// TIA Portal V20 export
FUNCTION_BLOCK "Sequence_3_TopTapeFixStage"   // FB32850, LAD
TITLE = Sequence
// Sequence template programmend in ladder logic
// stored: IsIECCheckEnabled true, MemoryReserve 100, Namespace Unit1.Em3, SetENOAutomatically true
   VAR_INPUT
      unitStatus : "LAF_typeUnitStatus";
   END_VAR
   VAR
      instSequenceLADControl { ExternalWritable := 'False'} : "LAF_ControlLadSequence";
      instSequenceLADStatus { ExternalWritable := 'False'} : "LAF_StatusLadSequence";
      statTonTime { ExternalWritable := 'False'} : Array[0..9999] of TON_TIME;
   END_VAR
   VAR_TEMP
      tempCustomerAction : Bool;   // Placeholder for possible actions
      tempDo_nothing_and_wait_for_init : Bool;   // Placeholder for doing nothing
      tempSafeStateCondition : Bool;   // Temp Condition for the equipment module to be in a safe state
   END_VAR
   VAR CONSTANT
      delayTime : Time := T#100ms;
      STEP_IDLE : DInt := 1;
      JOB_1_STEP_01 : DInt := 101;
      JOB_1_STEP_10 : DInt := 110;
      JOB_1_STEP_11 : DInt := 111;
      JOB_1_STEP_20 : DInt := 120;
      JOB_1_STEP_21 : DInt := 121;
      JOB_1_STEP_30 : DInt := 130;
      JOB_1_STEP_40 : DInt := 140;
      JOB_1_STEP_50 : DInt := 150;
      JOB_1_STEP_60 : DInt := 160;
      JOB_1_STEP_70 : DInt := 170;
      JOB_1_STEP_80 : DInt := 180;
      JOB_1_STEP_90 : DInt := 190;
      JOB_2_STEP_01 : DInt := 201;
      JOB_2_STEP_10 : DInt := 210;
      JOB_2_STEP_20 : DInt := 220;
      JOB_2_STEP_30 : DInt := 230;
      JOB_2_STEP_31 : DInt := 231;
      JOB_2_STEP_32 : DInt := 232;
      JOB_2_STEP_33 : DInt := 233;
      JOB_2_STEP_40 : DInt := 240;
      JOB_2_STEP_50 : DInt := 250;
      JOB_2_STEP_51 : DInt := 250;
      JOB_2_STEP_60 : DInt := 260;
      JOB_2_STEP_70 : DInt := 270;
      JOB_2_STEP_80 : DInt := 280;
      JOB_2_STEP_81 : DInt := 281;
      JOB_2_STEP_90 : DInt := 290;
      JOB_3_STEP_01 : DInt := 301;
      JOB_3_STEP_10 : DInt := 310;
      JOB_3_STEP_20 : DInt := 320;
      JOB_3_STEP_30 : DInt := 330;
      JOB_3_STEP_40 : DInt := 340;
      JOB_3_STEP_50 : DInt := 350;
      JOB_3_STEP_60 : DInt := 360;
      JOB_3_STEP_61 : DInt := 361;
      JOB_3_STEP_70 : DInt := 370;
      JOB_3_STEP_80 : DInt := 380;
      JOB_3_STEP_90 : DInt := 390;
      JOB_4_STEP_01 : DInt := 401;
      JOB_4_STEP_10 : DInt := 410;
      JOB_4_STEP_20 : DInt := 420;
      JOB_4_STEP_30 : DInt := 430;
      JOB_4_STEP_31 : DInt := 431;
      JOB_4_STEP_32 : DInt := 432;
      JOB_4_STEP_40 : DInt := 440;
      JOB_4_STEP_41 : DInt := 441;
      JOB_4_STEP_50 : DInt := 450;
      JOB_4_STEP_60 : DInt := 460;
      JOB_4_STEP_70 : DInt := 470;
      JOB_4_STEP_80 : DInt := 480;
      JOB_4_STEP_90 : DInt := 490;
      JOB_5_STEP_01 : DInt := 501;
      JOB_5_STEP_10 : DInt := 510;
      JOB_5_STEP_20 : DInt := 520;
      JOB_5_STEP_30 : DInt := 530;
      JOB_5_STEP_31 : DInt := 531;
      JOB_5_STEP_32 : DInt := 532;
      JOB_5_STEP_40 : DInt := 540;
      JOB_5_STEP_50 : DInt := 550;
      JOB_5_STEP_60 : DInt := 560;
      JOB_5_STEP_70 : DInt := 570;
      JOB_5_STEP_80 : DInt := 580;
      JOB_5_STEP_90 : DInt := 590;
      STEP_IMMEDIATE_STOP : DInt := 9001;   // Step executed when an immediate stop command is triggered for the sequence (i.e. when unit is in state aborting)
      TO_DO_INSERT_ACTIONS_HERE : Bool := TRUE;   // Template : Add actions
      TO_DO_INSERT_CONDITION_FOR_TRANSITION_HERE : Bool := TRUE;   // Template : Add conditions
   END_VAR
   VAR_TEMP   // added for the SCL form of the ladder/FBD networks
      _w1 : Bool;
      _w2 : Bool;
      _w3 : Bool;
   END_VAR
BEGIN

REGION Network 1: DESCRIPTION
   // This is a template block provided by the Automation Framework. It can be used to create an own project.
   // The Block Info Header is prepared to put in your own data.
   // Description of the block could be added here and the docu created by Code2Docu.
END_REGION

REGION Network 2: *************** CONTROL **********************
END_REGION

REGION Network 3: Sequence Control ("Enter your Sequins number here")
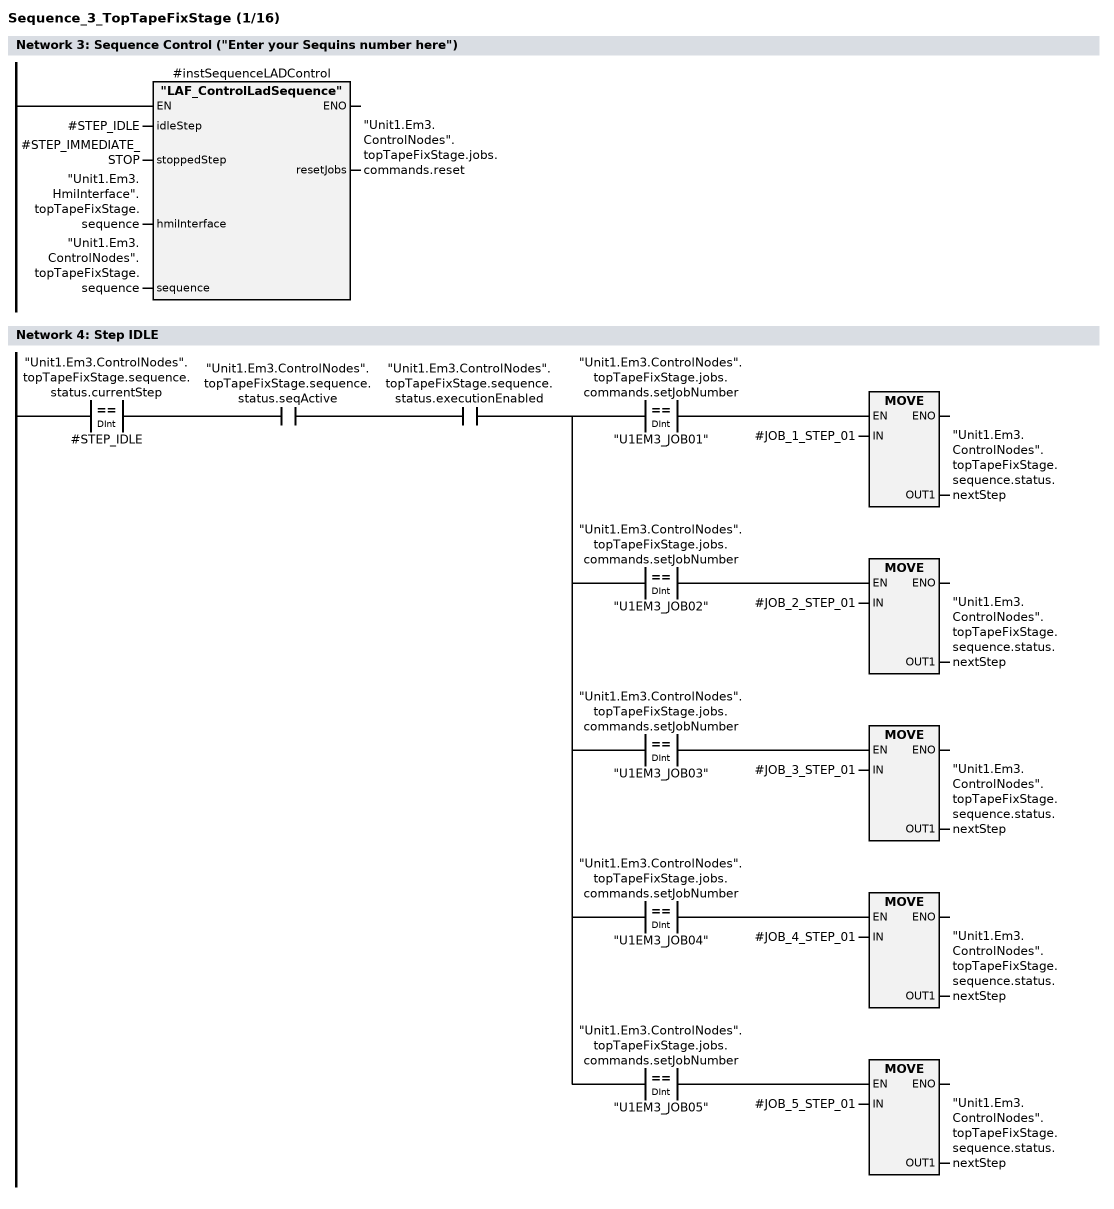
   RUNG wire#powerrail
      #instSequenceLADControl(idleStep := #STEP_IDLE, stoppedStep := #STEP_IMMEDIATE_STOP, hmiInterface := "Unit1.Em3.HmiInterface".topTapeFixStage.sequence, sequence := "Unit1.Em3.ControlNodes".topTapeFixStage.sequence, resetJobs => "Unit1.Em3.ControlNodes".topTapeFixStage.jobs.commands.reset)
   END_RUNG
   // the same network as SCL:
   #instSequenceLADControl(idleStep := #STEP_IDLE,   // "LAF_ControlLadSequence"
                           stoppedStep := #STEP_IMMEDIATE_STOP,
                           hmiInterface := "Unit1.Em3.HmiInterface".topTapeFixStage.sequence,
                           sequence := "Unit1.Em3.ControlNodes".topTapeFixStage.sequence,
                           resetJobs => "Unit1.Em3.ControlNodes".topTapeFixStage.jobs.commands.reset);
END_REGION

REGION Network 4: Step IDLE
   RUNG wire#powerrail
      { S7_Templates := "SrcType := DInt" } EQ_Contact(in1 := "Unit1.Em3.ControlNodes".topTapeFixStage.sequence.status.currentStep, in2 := #STEP_IDLE)
      Contact( "Unit1.Em3.ControlNodes".topTapeFixStage.sequence.status.seqActive )
      Contact( "Unit1.Em3.ControlNodes".topTapeFixStage.sequence.status.executionEnabled )
      wire#w1
      { S7_Templates := "SrcType := DInt" } EQ_Contact(in1 := "Unit1.Em3.ControlNodes".topTapeFixStage.jobs.commands.setJobNumber, in2 := "U1EM3_JOB01")
      Move(in := #JOB_1_STEP_01, out1 => "Unit1.Em3.ControlNodes".topTapeFixStage.sequence.status.nextStep)
   END_RUNG
   RUNG wire#w1
      { S7_Templates := "SrcType := DInt" } EQ_Contact(in1 := "Unit1.Em3.ControlNodes".topTapeFixStage.jobs.commands.setJobNumber, in2 := "U1EM3_JOB02")
      Move(in := #JOB_2_STEP_01, out1 => "Unit1.Em3.ControlNodes".topTapeFixStage.sequence.status.nextStep)
   END_RUNG
   RUNG wire#w1
      { S7_Templates := "SrcType := DInt" } EQ_Contact(in1 := "Unit1.Em3.ControlNodes".topTapeFixStage.jobs.commands.setJobNumber, in2 := "U1EM3_JOB03")
      Move(in := #JOB_3_STEP_01, out1 => "Unit1.Em3.ControlNodes".topTapeFixStage.sequence.status.nextStep)
   END_RUNG
   RUNG wire#w1
      { S7_Templates := "SrcType := DInt" } EQ_Contact(in1 := "Unit1.Em3.ControlNodes".topTapeFixStage.jobs.commands.setJobNumber, in2 := "U1EM3_JOB04")
      Move(in := #JOB_4_STEP_01, out1 => "Unit1.Em3.ControlNodes".topTapeFixStage.sequence.status.nextStep)
   END_RUNG
   RUNG wire#w1
      { S7_Templates := "SrcType := DInt" } EQ_Contact(in1 := "Unit1.Em3.ControlNodes".topTapeFixStage.jobs.commands.setJobNumber, in2 := "U1EM3_JOB05")
      Move(in := #JOB_5_STEP_01, out1 => "Unit1.Em3.ControlNodes".topTapeFixStage.sequence.status.nextStep)
   END_RUNG
   // the same network as SCL:
   #_w1 := ("Unit1.Em3.ControlNodes".topTapeFixStage.sequence.status.currentStep = #STEP_IDLE) AND "Unit1.Em3.ControlNodes".topTapeFixStage.sequence.status.seqActive AND "Unit1.Em3.ControlNodes".topTapeFixStage.sequence.status.executionEnabled;
   IF #_w1 AND ("Unit1.Em3.ControlNodes".topTapeFixStage.jobs.commands.setJobNumber = "U1EM3_JOB01") THEN
       "Unit1.Em3.ControlNodes".topTapeFixStage.sequence.status.nextStep := #JOB_1_STEP_01;
   END_IF;
   IF #_w1 AND ("Unit1.Em3.ControlNodes".topTapeFixStage.jobs.commands.setJobNumber = "U1EM3_JOB02") THEN
       "Unit1.Em3.ControlNodes".topTapeFixStage.sequence.status.nextStep := #JOB_2_STEP_01;
   END_IF;
   IF #_w1 AND ("Unit1.Em3.ControlNodes".topTapeFixStage.jobs.commands.setJobNumber = "U1EM3_JOB03") THEN
       "Unit1.Em3.ControlNodes".topTapeFixStage.sequence.status.nextStep := #JOB_3_STEP_01;
   END_IF;
   IF #_w1 AND ("Unit1.Em3.ControlNodes".topTapeFixStage.jobs.commands.setJobNumber = "U1EM3_JOB04") THEN
       "Unit1.Em3.ControlNodes".topTapeFixStage.sequence.status.nextStep := #JOB_4_STEP_01;
   END_IF;
   IF #_w1 AND ("Unit1.Em3.ControlNodes".topTapeFixStage.jobs.commands.setJobNumber = "U1EM3_JOB05") THEN
       "Unit1.Em3.ControlNodes".topTapeFixStage.sequence.status.nextStep := #JOB_5_STEP_01;
   END_IF;
END_REGION

REGION Network 6: *************** JOB[1] EM HOMING *************************
END_REGION

REGION Network 7: Step[101] : JOB[1] Condition
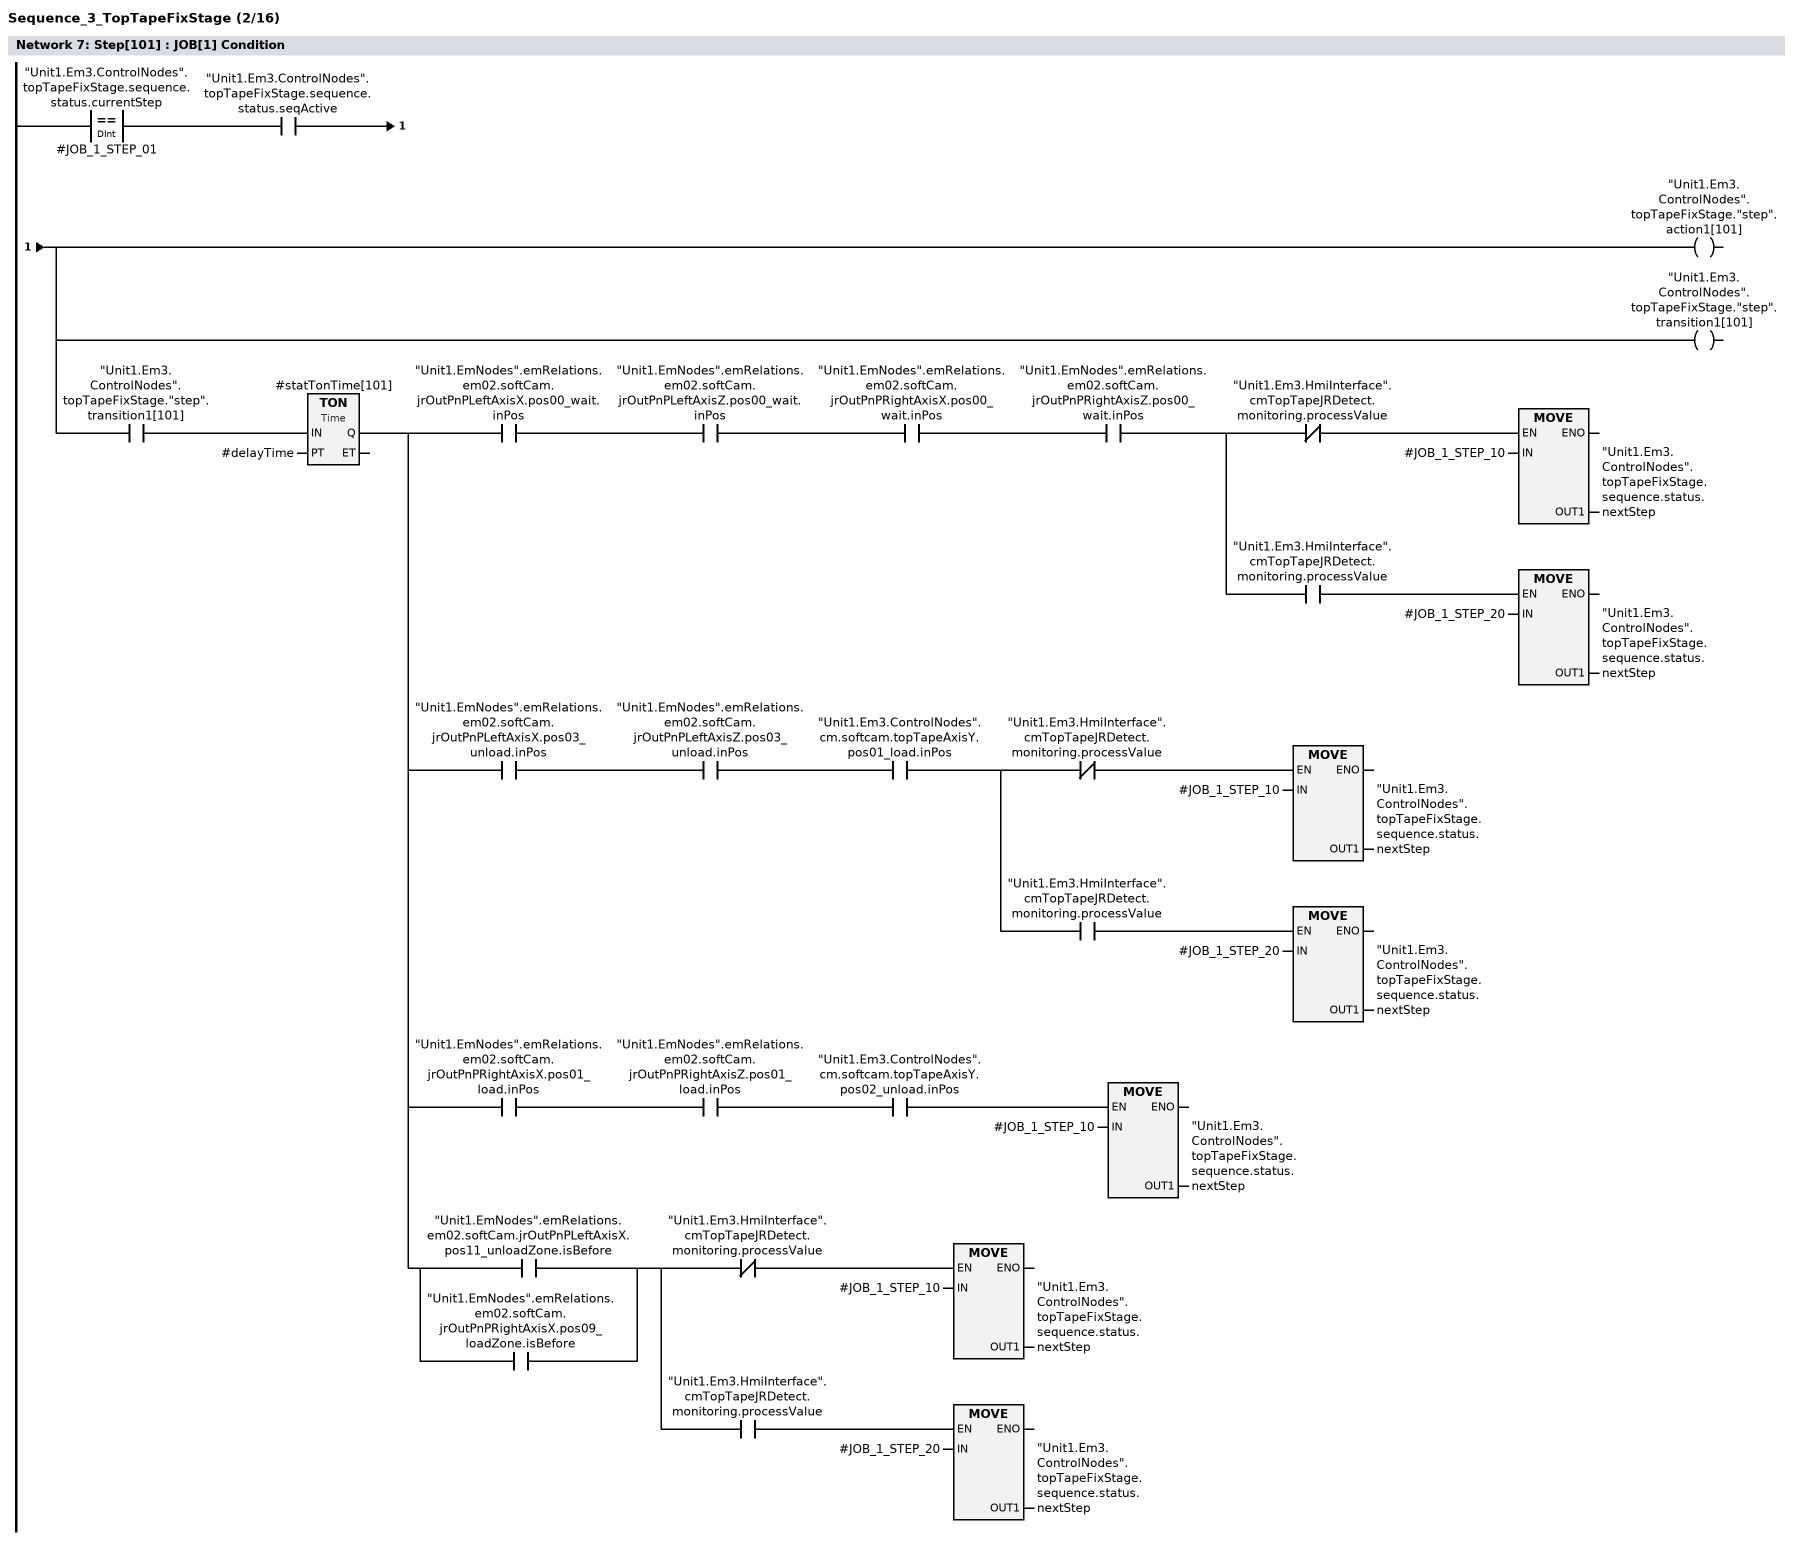
   RUNG wire#powerrail
      { S7_Templates := "SrcType := DInt" } EQ_Contact(in1 := "Unit1.Em3.ControlNodes".topTapeFixStage.sequence.status.currentStep, in2 := #JOB_1_STEP_01)
      Contact( "Unit1.Em3.ControlNodes".topTapeFixStage.sequence.status.seqActive )
      wire#w1
      Coil( "Unit1.Em3.ControlNodes".topTapeFixStage."step".action1[101] )
   END_RUNG
   RUNG wire#w1
      Coil( "Unit1.Em3.ControlNodes".topTapeFixStage."step".transition1[101] )
   END_RUNG
   RUNG wire#w1
      Contact( "Unit1.Em3.ControlNodes".topTapeFixStage."step".transition1[101] )
      { S7_Templates := "time_type := Time" } #statTonTime[101].TON(pt := #delayTime, et =>)
      wire#w2
      Contact( "Unit1.EmNodes".emRelations.em02.softCam.jrOutPnPLeftAxisX.pos00_wait.inPos )
      Contact( "Unit1.EmNodes".emRelations.em02.softCam.jrOutPnPLeftAxisZ.pos00_wait.inPos )
      Contact( "Unit1.EmNodes".emRelations.em02.softCam.jrOutPnPRightAxisX.pos00_wait.inPos )
      Contact( "Unit1.EmNodes".emRelations.em02.softCam.jrOutPnPRightAxisZ.pos00_wait.inPos )
      wire#w3
      I_Contact( "Unit1.Em3.HmiInterface".cmTopTapeJRDetect.monitoring.processValue )
      Move(in := #JOB_1_STEP_10, out1 => "Unit1.Em3.ControlNodes".topTapeFixStage.sequence.status.nextStep)
   END_RUNG
   RUNG wire#w3
      Contact( "Unit1.Em3.HmiInterface".cmTopTapeJRDetect.monitoring.processValue )
      Move(in := #JOB_1_STEP_20, out1 => "Unit1.Em3.ControlNodes".topTapeFixStage.sequence.status.nextStep)
   END_RUNG
   RUNG wire#w2
      Contact( "Unit1.EmNodes".emRelations.em02.softCam.jrOutPnPLeftAxisX.pos03_unload.inPos )
      Contact( "Unit1.EmNodes".emRelations.em02.softCam.jrOutPnPLeftAxisZ.pos03_unload.inPos )
      Contact( "Unit1.Em3.ControlNodes".cm.softcam.topTapeAxisY.pos01_load.inPos )
      wire#w4
      I_Contact( "Unit1.Em3.HmiInterface".cmTopTapeJRDetect.monitoring.processValue )
      Move(in := #JOB_1_STEP_10, out1 => "Unit1.Em3.ControlNodes".topTapeFixStage.sequence.status.nextStep)
   END_RUNG
   RUNG wire#w4
      Contact( "Unit1.Em3.HmiInterface".cmTopTapeJRDetect.monitoring.processValue )
      Move(in := #JOB_1_STEP_20, out1 => "Unit1.Em3.ControlNodes".topTapeFixStage.sequence.status.nextStep)
   END_RUNG
   RUNG wire#w2
      Contact( "Unit1.EmNodes".emRelations.em02.softCam.jrOutPnPRightAxisX.pos01_load.inPos )
      Contact( "Unit1.EmNodes".emRelations.em02.softCam.jrOutPnPRightAxisZ.pos01_load.inPos )
      Contact( "Unit1.Em3.ControlNodes".cm.softcam.topTapeAxisY.pos02_unload.inPos )
      Move(in := #JOB_1_STEP_10, out1 => "Unit1.Em3.ControlNodes".topTapeFixStage.sequence.status.nextStep)
   END_RUNG
   RUNG wire#w2
      Contact( "Unit1.EmNodes".emRelations.em02.softCam.jrOutPnPLeftAxisX.pos11_unloadZone.isBefore )
      wire#w5
      I_Contact( "Unit1.Em3.HmiInterface".cmTopTapeJRDetect.monitoring.processValue )
      Move(in := #JOB_1_STEP_10, out1 => "Unit1.Em3.ControlNodes".topTapeFixStage.sequence.status.nextStep)
   END_RUNG
   RUNG wire#w2
      Contact( "Unit1.EmNodes".emRelations.em02.softCam.jrOutPnPRightAxisX.pos09_loadZone.isBefore )
   END_RUNG wire#w5
   RUNG wire#w5
      Contact( "Unit1.Em3.HmiInterface".cmTopTapeJRDetect.monitoring.processValue )
      Move(in := #JOB_1_STEP_20, out1 => "Unit1.Em3.ControlNodes".topTapeFixStage.sequence.status.nextStep)
   END_RUNG
   // the same network as SCL:
   "Unit1.Em3.ControlNodes".topTapeFixStage."step".action1[101] := ("Unit1.Em3.ControlNodes".topTapeFixStage.sequence.status.currentStep = #JOB_1_STEP_01) AND "Unit1.Em3.ControlNodes".topTapeFixStage.sequence.status.seqActive;
   "Unit1.Em3.ControlNodes".topTapeFixStage."step".transition1[101] := ("Unit1.Em3.ControlNodes".topTapeFixStage.sequence.status.currentStep = #JOB_1_STEP_01) AND "Unit1.Em3.ControlNodes".topTapeFixStage.sequence.status.seqActive;
   #statTonTime[101].TON(IN := ("Unit1.Em3.ControlNodes".topTapeFixStage.sequence.status.currentStep = #JOB_1_STEP_01) AND "Unit1.Em3.ControlNodes".topTapeFixStage.sequence.status.seqActive AND "Unit1.Em3.ControlNodes".topTapeFixStage."step".transition1[101],
                         PT := #delayTime);
   #_w1 := #statTonTime[101].Q AND "Unit1.EmNodes".emRelations.em02.softCam.jrOutPnPLeftAxisX.pos00_wait.inPos AND "Unit1.EmNodes".emRelations.em02.softCam.jrOutPnPLeftAxisZ.pos00_wait.inPos AND "Unit1.EmNodes".emRelations.em02.softCam.jrOutPnPRightAxisX.pos00_wait.inPos AND "Unit1.EmNodes".emRelations.em02.softCam.jrOutPnPRightAxisZ.pos00_wait.inPos;
   IF #_w1 AND NOT "Unit1.Em3.HmiInterface".cmTopTapeJRDetect.monitoring.processValue THEN
       "Unit1.Em3.ControlNodes".topTapeFixStage.sequence.status.nextStep := #JOB_1_STEP_10;
   END_IF;
   IF #_w1 AND "Unit1.Em3.HmiInterface".cmTopTapeJRDetect.monitoring.processValue THEN
       "Unit1.Em3.ControlNodes".topTapeFixStage.sequence.status.nextStep := #JOB_1_STEP_20;
   END_IF;
   #_w2 := #statTonTime[101].Q AND "Unit1.EmNodes".emRelations.em02.softCam.jrOutPnPLeftAxisX.pos03_unload.inPos AND "Unit1.EmNodes".emRelations.em02.softCam.jrOutPnPLeftAxisZ.pos03_unload.inPos AND "Unit1.Em3.ControlNodes".cm.softcam.topTapeAxisY.pos01_load.inPos;
   IF #_w2 AND NOT "Unit1.Em3.HmiInterface".cmTopTapeJRDetect.monitoring.processValue THEN
       "Unit1.Em3.ControlNodes".topTapeFixStage.sequence.status.nextStep := #JOB_1_STEP_10;
   END_IF;
   IF #_w2 AND "Unit1.Em3.HmiInterface".cmTopTapeJRDetect.monitoring.processValue THEN
       "Unit1.Em3.ControlNodes".topTapeFixStage.sequence.status.nextStep := #JOB_1_STEP_20;
   END_IF;
   IF #statTonTime[101].Q AND "Unit1.EmNodes".emRelations.em02.softCam.jrOutPnPRightAxisX.pos01_load.inPos AND "Unit1.EmNodes".emRelations.em02.softCam.jrOutPnPRightAxisZ.pos01_load.inPos AND "Unit1.Em3.ControlNodes".cm.softcam.topTapeAxisY.pos02_unload.inPos THEN
       "Unit1.Em3.ControlNodes".topTapeFixStage.sequence.status.nextStep := #JOB_1_STEP_10;
   END_IF;
   #_w3 := #statTonTime[101].Q AND ("Unit1.EmNodes".emRelations.em02.softCam.jrOutPnPLeftAxisX.pos11_unloadZone.isBefore OR "Unit1.EmNodes".emRelations.em02.softCam.jrOutPnPRightAxisX.pos09_loadZone.isBefore);
   IF #_w3 AND NOT "Unit1.Em3.HmiInterface".cmTopTapeJRDetect.monitoring.processValue THEN
       "Unit1.Em3.ControlNodes".topTapeFixStage.sequence.status.nextStep := #JOB_1_STEP_10;
   END_IF;
   IF #_w3 AND "Unit1.Em3.HmiInterface".cmTopTapeJRDetect.monitoring.processValue THEN
       "Unit1.Em3.ControlNodes".topTapeFixStage.sequence.status.nextStep := #JOB_1_STEP_20;
   END_IF;
END_REGION

REGION Network 8: Step[110] : Top Tape Fix Stage Left/Center/Right Top Clamp Up
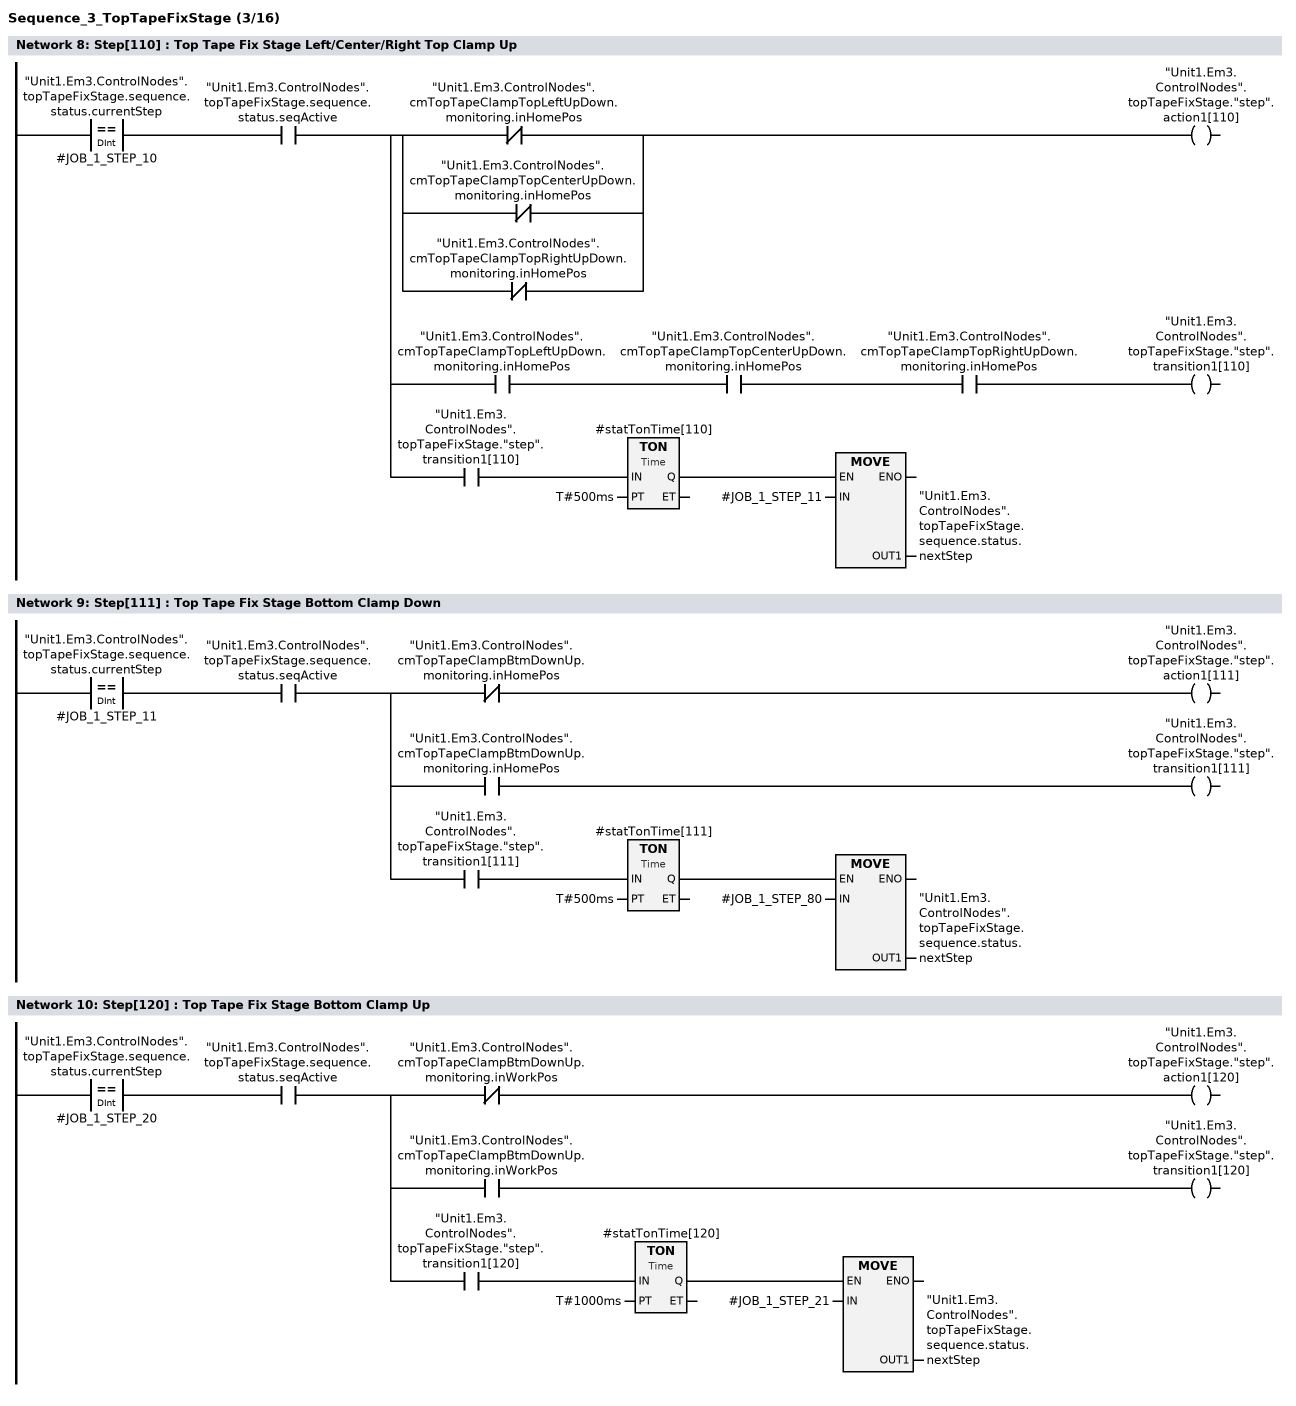
   RUNG wire#powerrail
      { S7_Templates := "SrcType := DInt" } EQ_Contact(in1 := "Unit1.Em3.ControlNodes".topTapeFixStage.sequence.status.currentStep, in2 := #JOB_1_STEP_10)
      Contact( "Unit1.Em3.ControlNodes".topTapeFixStage.sequence.status.seqActive )
      wire#w1
      I_Contact( "Unit1.Em3.ControlNodes".cmTopTapeClampTopLeftUpDown.monitoring.inHomePos )
      wire#w2
      Coil( "Unit1.Em3.ControlNodes".topTapeFixStage."step".action1[110] )
   END_RUNG
   RUNG wire#w1
      I_Contact( "Unit1.Em3.ControlNodes".cmTopTapeClampTopCenterUpDown.monitoring.inHomePos )
   END_RUNG wire#w2
   RUNG wire#w1
      I_Contact( "Unit1.Em3.ControlNodes".cmTopTapeClampTopRightUpDown.monitoring.inHomePos )
   END_RUNG wire#w2
   RUNG wire#w1
      Contact( "Unit1.Em3.ControlNodes".cmTopTapeClampTopLeftUpDown.monitoring.inHomePos )
      Contact( "Unit1.Em3.ControlNodes".cmTopTapeClampTopCenterUpDown.monitoring.inHomePos )
      Contact( "Unit1.Em3.ControlNodes".cmTopTapeClampTopRightUpDown.monitoring.inHomePos )
      Coil( "Unit1.Em3.ControlNodes".topTapeFixStage."step".transition1[110] )
   END_RUNG
   RUNG wire#w1
      Contact( "Unit1.Em3.ControlNodes".topTapeFixStage."step".transition1[110] )
      { S7_Templates := "time_type := Time" } #statTonTime[110].TON(pt := T#500ms, et =>)
      Move(in := #JOB_1_STEP_11, out1 => "Unit1.Em3.ControlNodes".topTapeFixStage.sequence.status.nextStep)
   END_RUNG
   // the same network as SCL:
   #_w1 := ("Unit1.Em3.ControlNodes".topTapeFixStage.sequence.status.currentStep = #JOB_1_STEP_10) AND "Unit1.Em3.ControlNodes".topTapeFixStage.sequence.status.seqActive;
   "Unit1.Em3.ControlNodes".topTapeFixStage."step".action1[110] := #_w1 AND (NOT "Unit1.Em3.ControlNodes".cmTopTapeClampTopLeftUpDown.monitoring.inHomePos OR NOT "Unit1.Em3.ControlNodes".cmTopTapeClampTopCenterUpDown.monitoring.inHomePos OR NOT "Unit1.Em3.ControlNodes".cmTopTapeClampTopRightUpDown.monitoring.inHomePos);
   "Unit1.Em3.ControlNodes".topTapeFixStage."step".transition1[110] := #_w1 AND "Unit1.Em3.ControlNodes".cmTopTapeClampTopLeftUpDown.monitoring.inHomePos AND "Unit1.Em3.ControlNodes".cmTopTapeClampTopCenterUpDown.monitoring.inHomePos AND "Unit1.Em3.ControlNodes".cmTopTapeClampTopRightUpDown.monitoring.inHomePos;
   #statTonTime[110].TON(IN := #_w1 AND "Unit1.Em3.ControlNodes".topTapeFixStage."step".transition1[110],
                         PT := T#500ms);
   IF #statTonTime[110].Q THEN
       "Unit1.Em3.ControlNodes".topTapeFixStage.sequence.status.nextStep := #JOB_1_STEP_11;
   END_IF;
END_REGION

REGION Network 9: Step[111] : Top Tape Fix Stage Bottom Clamp Down
   RUNG wire#powerrail
      { S7_Templates := "SrcType := DInt" } EQ_Contact(in1 := "Unit1.Em3.ControlNodes".topTapeFixStage.sequence.status.currentStep, in2 := #JOB_1_STEP_11)
      Contact( "Unit1.Em3.ControlNodes".topTapeFixStage.sequence.status.seqActive )
      wire#w1
      I_Contact( "Unit1.Em3.ControlNodes".cmTopTapeClampBtmDownUp.monitoring.inHomePos )
      Coil( "Unit1.Em3.ControlNodes".topTapeFixStage."step".action1[111] )
   END_RUNG
   RUNG wire#w1
      Contact( "Unit1.Em3.ControlNodes".cmTopTapeClampBtmDownUp.monitoring.inHomePos )
      Coil( "Unit1.Em3.ControlNodes".topTapeFixStage."step".transition1[111] )
   END_RUNG
   RUNG wire#w1
      Contact( "Unit1.Em3.ControlNodes".topTapeFixStage."step".transition1[111] )
      { S7_Templates := "time_type := Time" } #statTonTime[111].TON(pt := T#500ms, et =>)
      Move(in := #JOB_1_STEP_80, out1 => "Unit1.Em3.ControlNodes".topTapeFixStage.sequence.status.nextStep)
   END_RUNG
   // the same network as SCL:
   #_w1 := ("Unit1.Em3.ControlNodes".topTapeFixStage.sequence.status.currentStep = #JOB_1_STEP_11) AND "Unit1.Em3.ControlNodes".topTapeFixStage.sequence.status.seqActive;
   "Unit1.Em3.ControlNodes".topTapeFixStage."step".action1[111] := #_w1 AND NOT "Unit1.Em3.ControlNodes".cmTopTapeClampBtmDownUp.monitoring.inHomePos;
   "Unit1.Em3.ControlNodes".topTapeFixStage."step".transition1[111] := #_w1 AND "Unit1.Em3.ControlNodes".cmTopTapeClampBtmDownUp.monitoring.inHomePos;
   #statTonTime[111].TON(IN := #_w1 AND "Unit1.Em3.ControlNodes".topTapeFixStage."step".transition1[111],
                         PT := T#500ms);
   IF #statTonTime[111].Q THEN
       "Unit1.Em3.ControlNodes".topTapeFixStage.sequence.status.nextStep := #JOB_1_STEP_80;
   END_IF;
END_REGION

REGION Network 10: Step[120] : Top Tape Fix Stage Bottom Clamp Up
   RUNG wire#powerrail
      { S7_Templates := "SrcType := DInt" } EQ_Contact(in1 := "Unit1.Em3.ControlNodes".topTapeFixStage.sequence.status.currentStep, in2 := #JOB_1_STEP_20)
      Contact( "Unit1.Em3.ControlNodes".topTapeFixStage.sequence.status.seqActive )
      wire#w1
      I_Contact( "Unit1.Em3.ControlNodes".cmTopTapeClampBtmDownUp.monitoring.inWorkPos )
      Coil( "Unit1.Em3.ControlNodes".topTapeFixStage."step".action1[120] )
   END_RUNG
   RUNG wire#w1
      Contact( "Unit1.Em3.ControlNodes".cmTopTapeClampBtmDownUp.monitoring.inWorkPos )
      Coil( "Unit1.Em3.ControlNodes".topTapeFixStage."step".transition1[120] )
   END_RUNG
   RUNG wire#w1
      Contact( "Unit1.Em3.ControlNodes".topTapeFixStage."step".transition1[120] )
      { S7_Templates := "time_type := Time" } #statTonTime[120].TON(pt := T#1000ms, et =>)
      Move(in := #JOB_1_STEP_21, out1 => "Unit1.Em3.ControlNodes".topTapeFixStage.sequence.status.nextStep)
   END_RUNG
   // the same network as SCL:
   #_w1 := ("Unit1.Em3.ControlNodes".topTapeFixStage.sequence.status.currentStep = #JOB_1_STEP_20) AND "Unit1.Em3.ControlNodes".topTapeFixStage.sequence.status.seqActive;
   "Unit1.Em3.ControlNodes".topTapeFixStage."step".action1[120] := #_w1 AND NOT "Unit1.Em3.ControlNodes".cmTopTapeClampBtmDownUp.monitoring.inWorkPos;
   "Unit1.Em3.ControlNodes".topTapeFixStage."step".transition1[120] := #_w1 AND "Unit1.Em3.ControlNodes".cmTopTapeClampBtmDownUp.monitoring.inWorkPos;
   #statTonTime[120].TON(IN := #_w1 AND "Unit1.Em3.ControlNodes".topTapeFixStage."step".transition1[120],
                         PT := T#1000ms);
   IF #statTonTime[120].Q THEN
       "Unit1.Em3.ControlNodes".topTapeFixStage.sequence.status.nextStep := #JOB_1_STEP_21;
   END_IF;
END_REGION

REGION Network 11: Step[121] : Top Tape Fix Stage Left/Center/Right Top Clamp Down
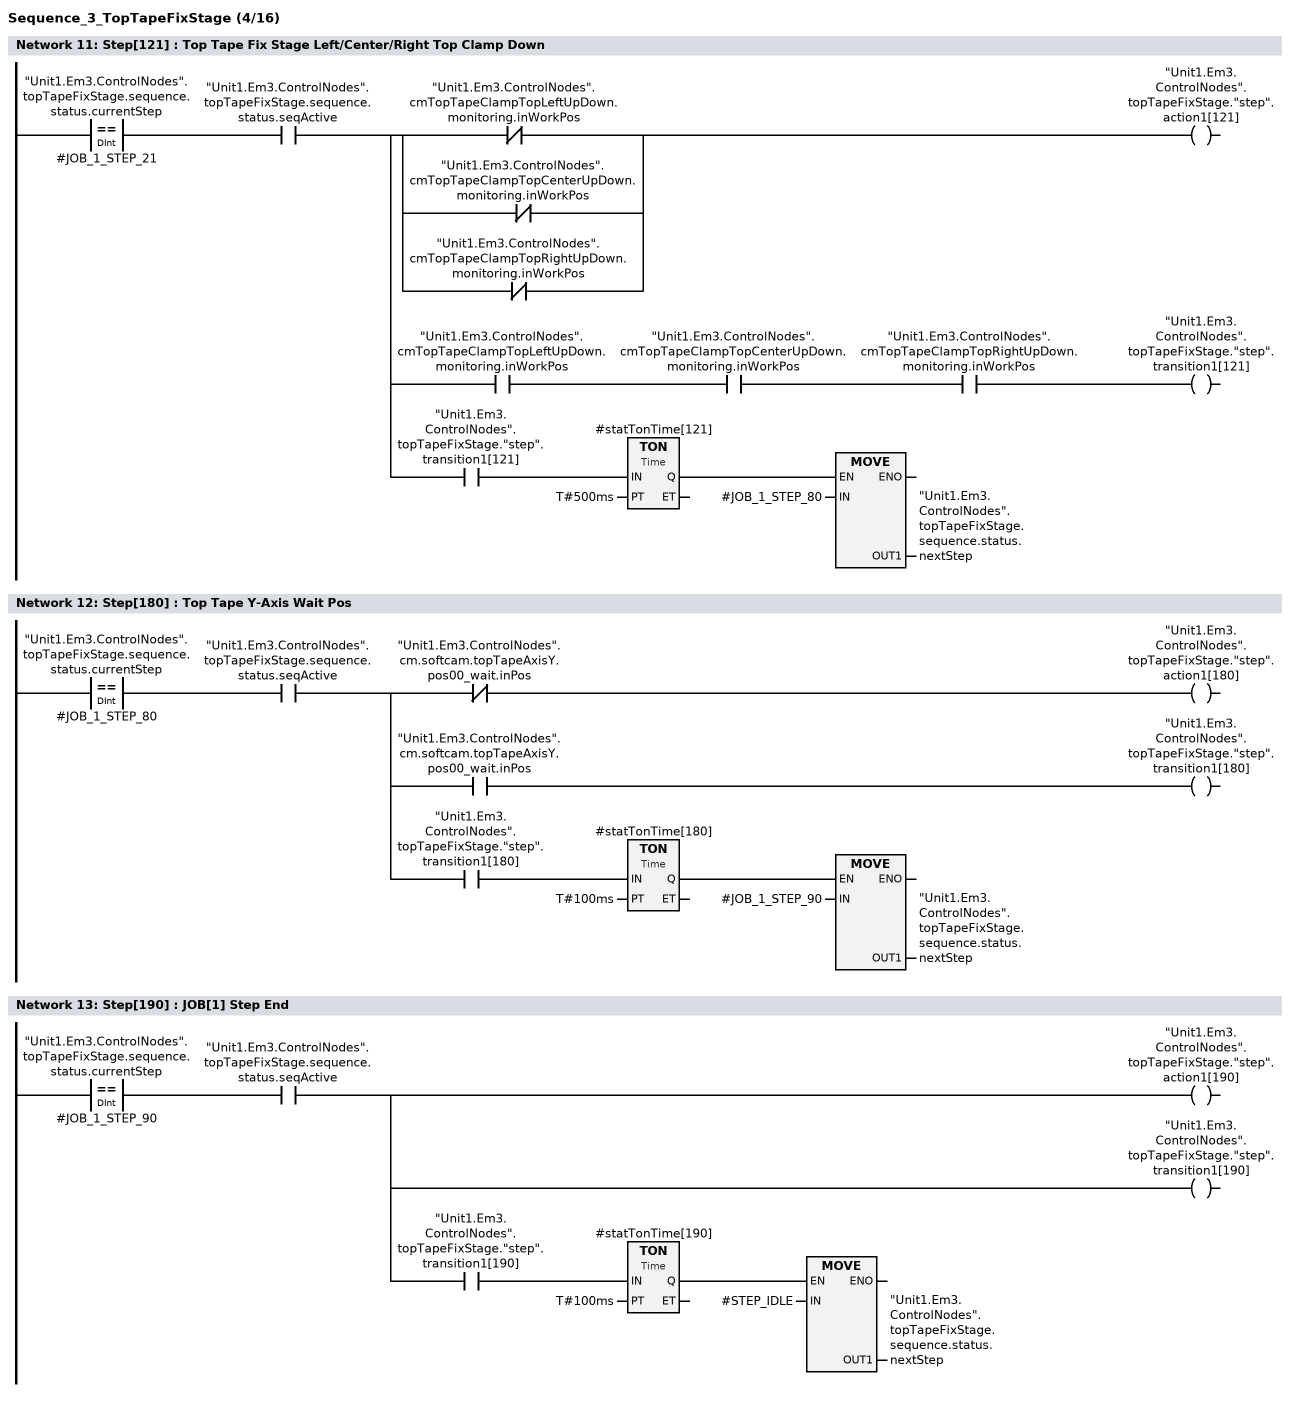
   RUNG wire#powerrail
      { S7_Templates := "SrcType := DInt" } EQ_Contact(in1 := "Unit1.Em3.ControlNodes".topTapeFixStage.sequence.status.currentStep, in2 := #JOB_1_STEP_21)
      Contact( "Unit1.Em3.ControlNodes".topTapeFixStage.sequence.status.seqActive )
      wire#w1
      I_Contact( "Unit1.Em3.ControlNodes".cmTopTapeClampTopLeftUpDown.monitoring.inWorkPos )
      wire#w2
      Coil( "Unit1.Em3.ControlNodes".topTapeFixStage."step".action1[121] )
   END_RUNG
   RUNG wire#w1
      I_Contact( "Unit1.Em3.ControlNodes".cmTopTapeClampTopCenterUpDown.monitoring.inWorkPos )
   END_RUNG wire#w2
   RUNG wire#w1
      I_Contact( "Unit1.Em3.ControlNodes".cmTopTapeClampTopRightUpDown.monitoring.inWorkPos )
   END_RUNG wire#w2
   RUNG wire#w1
      Contact( "Unit1.Em3.ControlNodes".cmTopTapeClampTopLeftUpDown.monitoring.inWorkPos )
      Contact( "Unit1.Em3.ControlNodes".cmTopTapeClampTopCenterUpDown.monitoring.inWorkPos )
      Contact( "Unit1.Em3.ControlNodes".cmTopTapeClampTopRightUpDown.monitoring.inWorkPos )
      Coil( "Unit1.Em3.ControlNodes".topTapeFixStage."step".transition1[121] )
   END_RUNG
   RUNG wire#w1
      Contact( "Unit1.Em3.ControlNodes".topTapeFixStage."step".transition1[121] )
      { S7_Templates := "time_type := Time" } #statTonTime[121].TON(pt := T#500ms, et =>)
      Move(in := #JOB_1_STEP_80, out1 => "Unit1.Em3.ControlNodes".topTapeFixStage.sequence.status.nextStep)
   END_RUNG
   // the same network as SCL:
   #_w1 := ("Unit1.Em3.ControlNodes".topTapeFixStage.sequence.status.currentStep = #JOB_1_STEP_21) AND "Unit1.Em3.ControlNodes".topTapeFixStage.sequence.status.seqActive;
   "Unit1.Em3.ControlNodes".topTapeFixStage."step".action1[121] := #_w1 AND (NOT "Unit1.Em3.ControlNodes".cmTopTapeClampTopLeftUpDown.monitoring.inWorkPos OR NOT "Unit1.Em3.ControlNodes".cmTopTapeClampTopCenterUpDown.monitoring.inWorkPos OR NOT "Unit1.Em3.ControlNodes".cmTopTapeClampTopRightUpDown.monitoring.inWorkPos);
   "Unit1.Em3.ControlNodes".topTapeFixStage."step".transition1[121] := #_w1 AND "Unit1.Em3.ControlNodes".cmTopTapeClampTopLeftUpDown.monitoring.inWorkPos AND "Unit1.Em3.ControlNodes".cmTopTapeClampTopCenterUpDown.monitoring.inWorkPos AND "Unit1.Em3.ControlNodes".cmTopTapeClampTopRightUpDown.monitoring.inWorkPos;
   #statTonTime[121].TON(IN := #_w1 AND "Unit1.Em3.ControlNodes".topTapeFixStage."step".transition1[121],
                         PT := T#500ms);
   IF #statTonTime[121].Q THEN
       "Unit1.Em3.ControlNodes".topTapeFixStage.sequence.status.nextStep := #JOB_1_STEP_80;
   END_IF;
END_REGION

REGION Network 12: Step[180] : Top Tape Y-Axis Wait Pos
   RUNG wire#powerrail
      { S7_Templates := "SrcType := DInt" } EQ_Contact(in1 := "Unit1.Em3.ControlNodes".topTapeFixStage.sequence.status.currentStep, in2 := #JOB_1_STEP_80)
      Contact( "Unit1.Em3.ControlNodes".topTapeFixStage.sequence.status.seqActive )
      wire#w1
      I_Contact( "Unit1.Em3.ControlNodes".cm.softcam.topTapeAxisY.pos00_wait.inPos )
      Coil( "Unit1.Em3.ControlNodes".topTapeFixStage."step".action1[180] )
   END_RUNG
   RUNG wire#w1
      Contact( "Unit1.Em3.ControlNodes".cm.softcam.topTapeAxisY.pos00_wait.inPos )
      Coil( "Unit1.Em3.ControlNodes".topTapeFixStage."step".transition1[180] )
   END_RUNG
   RUNG wire#w1
      Contact( "Unit1.Em3.ControlNodes".topTapeFixStage."step".transition1[180] )
      { S7_Templates := "time_type := Time" } #statTonTime[180].TON(pt := T#100ms, et =>)
      Move(in := #JOB_1_STEP_90, out1 => "Unit1.Em3.ControlNodes".topTapeFixStage.sequence.status.nextStep)
   END_RUNG
   // the same network as SCL:
   #_w1 := ("Unit1.Em3.ControlNodes".topTapeFixStage.sequence.status.currentStep = #JOB_1_STEP_80) AND "Unit1.Em3.ControlNodes".topTapeFixStage.sequence.status.seqActive;
   "Unit1.Em3.ControlNodes".topTapeFixStage."step".action1[180] := #_w1 AND NOT "Unit1.Em3.ControlNodes".cm.softcam.topTapeAxisY.pos00_wait.inPos;
   "Unit1.Em3.ControlNodes".topTapeFixStage."step".transition1[180] := #_w1 AND "Unit1.Em3.ControlNodes".cm.softcam.topTapeAxisY.pos00_wait.inPos;
   #statTonTime[180].TON(IN := #_w1 AND "Unit1.Em3.ControlNodes".topTapeFixStage."step".transition1[180],
                         PT := T#100ms);
   IF #statTonTime[180].Q THEN
       "Unit1.Em3.ControlNodes".topTapeFixStage.sequence.status.nextStep := #JOB_1_STEP_90;
   END_IF;
END_REGION

REGION Network 13: Step[190] : JOB[1] Step End
   RUNG wire#powerrail
      { S7_Templates := "SrcType := DInt" } EQ_Contact(in1 := "Unit1.Em3.ControlNodes".topTapeFixStage.sequence.status.currentStep, in2 := #JOB_1_STEP_90)
      Contact( "Unit1.Em3.ControlNodes".topTapeFixStage.sequence.status.seqActive )
      wire#w1
      Coil( "Unit1.Em3.ControlNodes".topTapeFixStage."step".action1[190] )
   END_RUNG
   RUNG wire#w1
      Coil( "Unit1.Em3.ControlNodes".topTapeFixStage."step".transition1[190] )
   END_RUNG
   RUNG wire#w1
      Contact( "Unit1.Em3.ControlNodes".topTapeFixStage."step".transition1[190] )
      { S7_Templates := "time_type := Time" } #statTonTime[190].TON(pt := T#100ms, et =>)
      Move(in := #STEP_IDLE, out1 => "Unit1.Em3.ControlNodes".topTapeFixStage.sequence.status.nextStep)
   END_RUNG
   // the same network as SCL:
   "Unit1.Em3.ControlNodes".topTapeFixStage."step".action1[190] := ("Unit1.Em3.ControlNodes".topTapeFixStage.sequence.status.currentStep = #JOB_1_STEP_90) AND "Unit1.Em3.ControlNodes".topTapeFixStage.sequence.status.seqActive;
   "Unit1.Em3.ControlNodes".topTapeFixStage."step".transition1[190] := ("Unit1.Em3.ControlNodes".topTapeFixStage.sequence.status.currentStep = #JOB_1_STEP_90) AND "Unit1.Em3.ControlNodes".topTapeFixStage.sequence.status.seqActive;
   #statTonTime[190].TON(IN := ("Unit1.Em3.ControlNodes".topTapeFixStage.sequence.status.currentStep = #JOB_1_STEP_90) AND "Unit1.Em3.ControlNodes".topTapeFixStage.sequence.status.seqActive AND "Unit1.Em3.ControlNodes".topTapeFixStage."step".transition1[190],
                         PT := T#100ms);
   IF #statTonTime[190].Q THEN
       "Unit1.Em3.ControlNodes".topTapeFixStage.sequence.status.nextStep := #STEP_IDLE;
   END_IF;
END_REGION

REGION Network 14: *************** JOB[2] JR GET=AUTO *************************
END_REGION

REGION Network 15: Step[201] : JOB[2] Condition
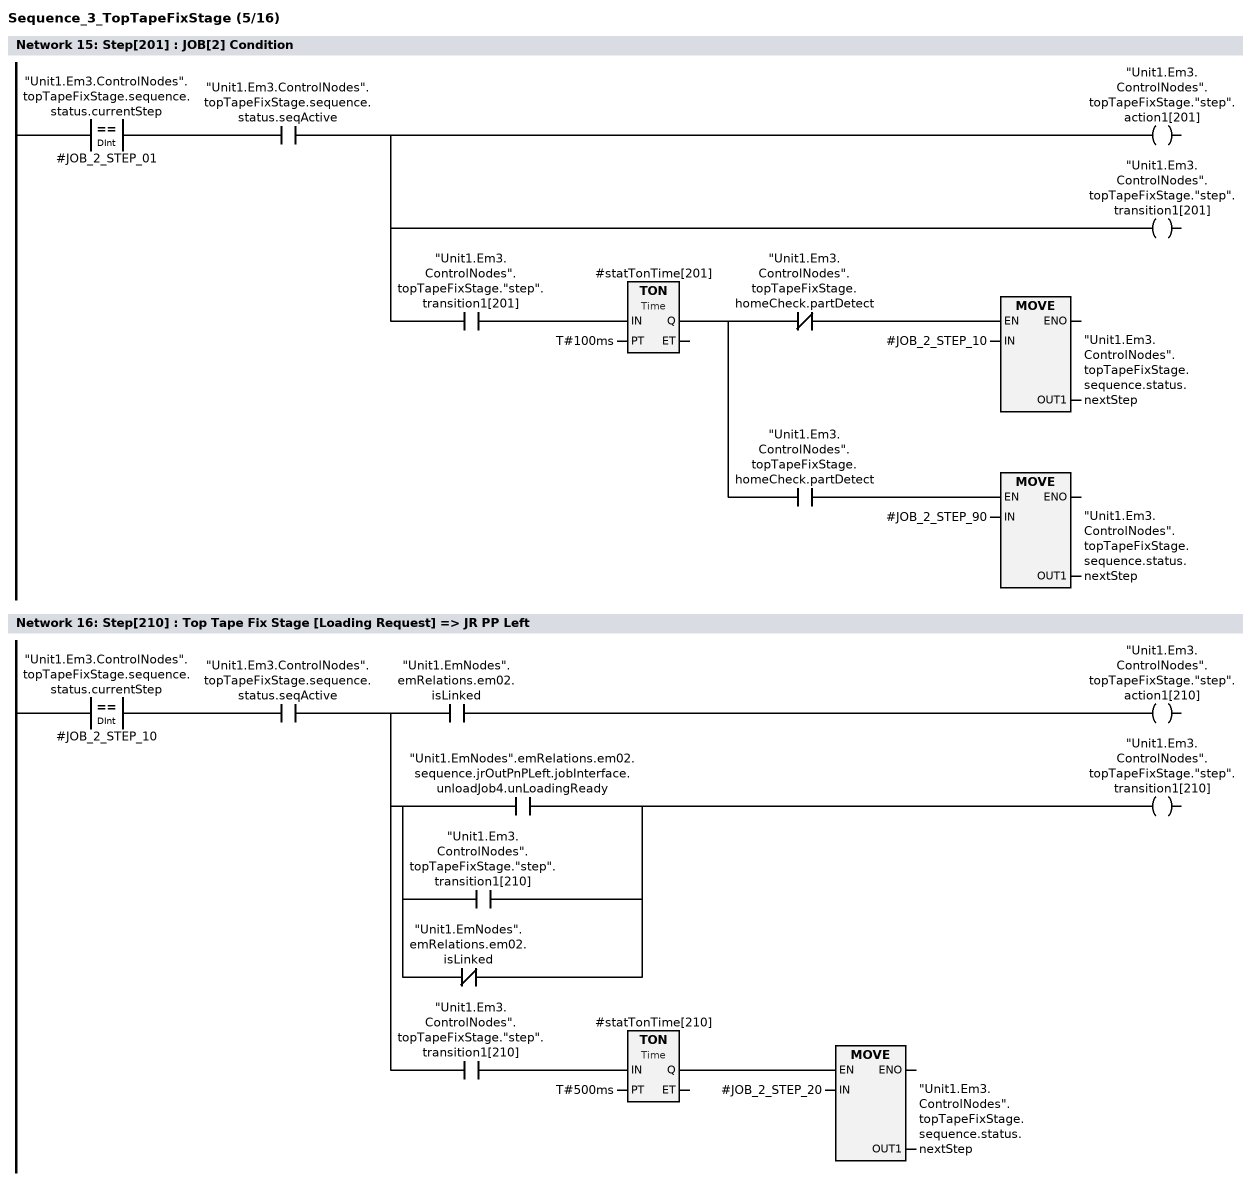
   RUNG wire#powerrail
      { S7_Templates := "SrcType := DInt" } EQ_Contact(in1 := "Unit1.Em3.ControlNodes".topTapeFixStage.sequence.status.currentStep, in2 := #JOB_2_STEP_01)
      Contact( "Unit1.Em3.ControlNodes".topTapeFixStage.sequence.status.seqActive )
      wire#w1
      Coil( "Unit1.Em3.ControlNodes".topTapeFixStage."step".action1[201] )
   END_RUNG
   RUNG wire#w1
      Coil( "Unit1.Em3.ControlNodes".topTapeFixStage."step".transition1[201] )
   END_RUNG
   RUNG wire#w1
      Contact( "Unit1.Em3.ControlNodes".topTapeFixStage."step".transition1[201] )
      { S7_Templates := "time_type := Time" } #statTonTime[201].TON(pt := T#100ms, et =>)
      wire#w2
      I_Contact( "Unit1.Em3.ControlNodes".topTapeFixStage.homeCheck.partDetect )
      Move(in := #JOB_2_STEP_10, out1 => "Unit1.Em3.ControlNodes".topTapeFixStage.sequence.status.nextStep)
   END_RUNG
   RUNG wire#w2
      Contact( "Unit1.Em3.ControlNodes".topTapeFixStage.homeCheck.partDetect )
      Move(in := #JOB_2_STEP_90, out1 => "Unit1.Em3.ControlNodes".topTapeFixStage.sequence.status.nextStep)
   END_RUNG
   // the same network as SCL:
   "Unit1.Em3.ControlNodes".topTapeFixStage."step".action1[201] := ("Unit1.Em3.ControlNodes".topTapeFixStage.sequence.status.currentStep = #JOB_2_STEP_01) AND "Unit1.Em3.ControlNodes".topTapeFixStage.sequence.status.seqActive;
   "Unit1.Em3.ControlNodes".topTapeFixStage."step".transition1[201] := ("Unit1.Em3.ControlNodes".topTapeFixStage.sequence.status.currentStep = #JOB_2_STEP_01) AND "Unit1.Em3.ControlNodes".topTapeFixStage.sequence.status.seqActive;
   #statTonTime[201].TON(IN := ("Unit1.Em3.ControlNodes".topTapeFixStage.sequence.status.currentStep = #JOB_2_STEP_01) AND "Unit1.Em3.ControlNodes".topTapeFixStage.sequence.status.seqActive AND "Unit1.Em3.ControlNodes".topTapeFixStage."step".transition1[201],
                         PT := T#100ms);
   IF #statTonTime[201].Q AND NOT "Unit1.Em3.ControlNodes".topTapeFixStage.homeCheck.partDetect THEN
       "Unit1.Em3.ControlNodes".topTapeFixStage.sequence.status.nextStep := #JOB_2_STEP_10;
   END_IF;
   IF #statTonTime[201].Q AND "Unit1.Em3.ControlNodes".topTapeFixStage.homeCheck.partDetect THEN
       "Unit1.Em3.ControlNodes".topTapeFixStage.sequence.status.nextStep := #JOB_2_STEP_90;
   END_IF;
END_REGION

REGION Network 16: Step[210] : Top Tape Fix Stage [Loading Request] => JR PP Left
   RUNG wire#powerrail
      { S7_Templates := "SrcType := DInt" } EQ_Contact(in1 := "Unit1.Em3.ControlNodes".topTapeFixStage.sequence.status.currentStep, in2 := #JOB_2_STEP_10)
      Contact( "Unit1.Em3.ControlNodes".topTapeFixStage.sequence.status.seqActive )
      wire#w1
      Contact( "Unit1.EmNodes".emRelations.em02.isLinked )
      Coil( "Unit1.Em3.ControlNodes".topTapeFixStage."step".action1[210] )
   END_RUNG
   RUNG wire#w1
      Contact( "Unit1.EmNodes".emRelations.em02.sequence.jrOutPnPLeft.jobInterface.unloadJob4.unLoadingReady )
      wire#w2
      Coil( "Unit1.Em3.ControlNodes".topTapeFixStage."step".transition1[210] )
   END_RUNG
   RUNG wire#w1
      Contact( "Unit1.Em3.ControlNodes".topTapeFixStage."step".transition1[210] )
   END_RUNG wire#w2
   RUNG wire#w1
      I_Contact( "Unit1.EmNodes".emRelations.em02.isLinked )
   END_RUNG wire#w2
   RUNG wire#w1
      Contact( "Unit1.Em3.ControlNodes".topTapeFixStage."step".transition1[210] )
      { S7_Templates := "time_type := Time" } #statTonTime[210].TON(pt := T#500ms, et =>)
      Move(in := #JOB_2_STEP_20, out1 => "Unit1.Em3.ControlNodes".topTapeFixStage.sequence.status.nextStep)
   END_RUNG
   // the same network as SCL:
   #_w1 := ("Unit1.Em3.ControlNodes".topTapeFixStage.sequence.status.currentStep = #JOB_2_STEP_10) AND "Unit1.Em3.ControlNodes".topTapeFixStage.sequence.status.seqActive;
   "Unit1.Em3.ControlNodes".topTapeFixStage."step".action1[210] := #_w1 AND "Unit1.EmNodes".emRelations.em02.isLinked;
   "Unit1.Em3.ControlNodes".topTapeFixStage."step".transition1[210] := #_w1 AND ("Unit1.EmNodes".emRelations.em02.sequence.jrOutPnPLeft.jobInterface.unloadJob4.unLoadingReady OR "Unit1.Em3.ControlNodes".topTapeFixStage."step".transition1[210] OR NOT "Unit1.EmNodes".emRelations.em02.isLinked);
   #statTonTime[210].TON(IN := #_w1 AND "Unit1.Em3.ControlNodes".topTapeFixStage."step".transition1[210],
                         PT := T#500ms);
   IF #statTonTime[210].Q THEN
       "Unit1.Em3.ControlNodes".topTapeFixStage.sequence.status.nextStep := #JOB_2_STEP_20;
   END_IF;
END_REGION

REGION Network 17: Step[220] Top Tape Y-Axis JR Put/Get Pos
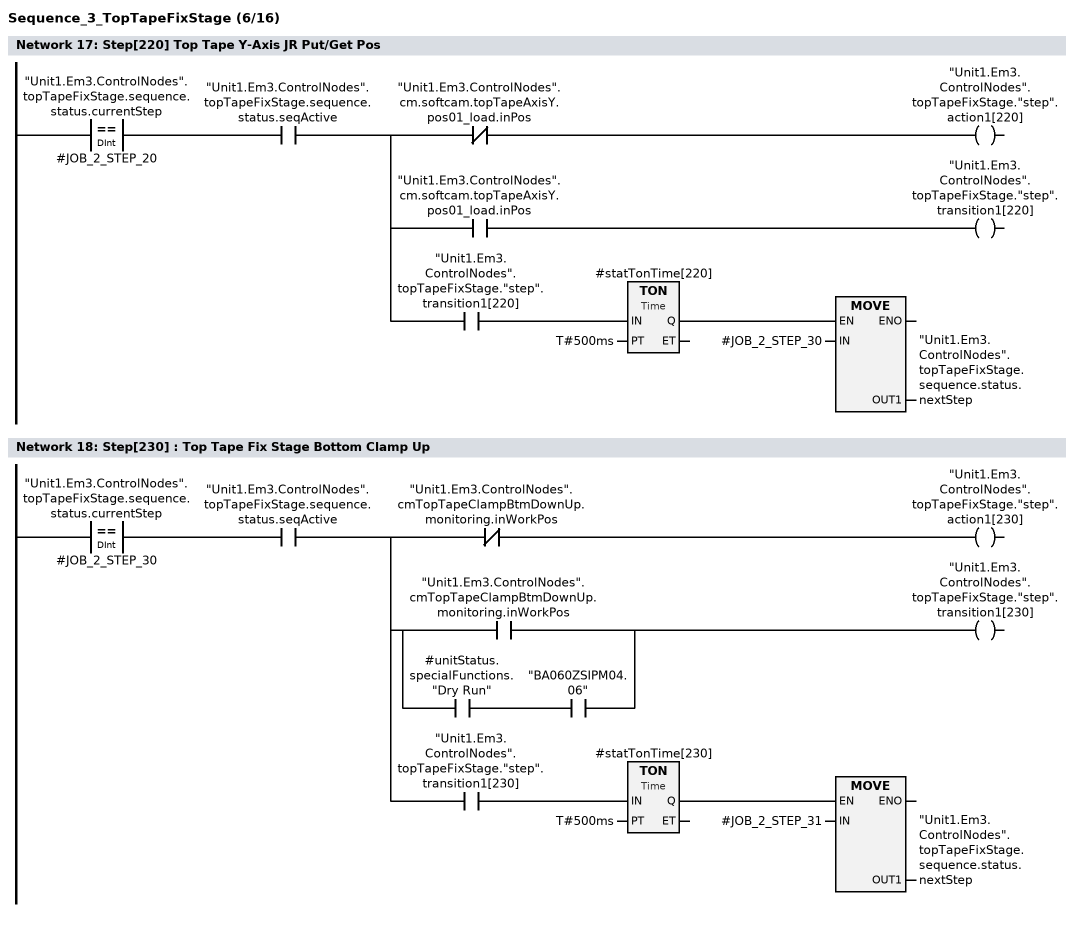
   RUNG wire#powerrail
      { S7_Templates := "SrcType := DInt" } EQ_Contact(in1 := "Unit1.Em3.ControlNodes".topTapeFixStage.sequence.status.currentStep, in2 := #JOB_2_STEP_20)
      Contact( "Unit1.Em3.ControlNodes".topTapeFixStage.sequence.status.seqActive )
      wire#w1
      I_Contact( "Unit1.Em3.ControlNodes".cm.softcam.topTapeAxisY.pos01_load.inPos )
      Coil( "Unit1.Em3.ControlNodes".topTapeFixStage."step".action1[220] )
   END_RUNG
   RUNG wire#w1
      Contact( "Unit1.Em3.ControlNodes".cm.softcam.topTapeAxisY.pos01_load.inPos )
      Coil( "Unit1.Em3.ControlNodes".topTapeFixStage."step".transition1[220] )
   END_RUNG
   RUNG wire#w1
      Contact( "Unit1.Em3.ControlNodes".topTapeFixStage."step".transition1[220] )
      { S7_Templates := "time_type := Time" } #statTonTime[220].TON(pt := T#500ms, et =>)
      Move(in := #JOB_2_STEP_30, out1 => "Unit1.Em3.ControlNodes".topTapeFixStage.sequence.status.nextStep)
   END_RUNG
   // the same network as SCL:
   #_w1 := ("Unit1.Em3.ControlNodes".topTapeFixStage.sequence.status.currentStep = #JOB_2_STEP_20) AND "Unit1.Em3.ControlNodes".topTapeFixStage.sequence.status.seqActive;
   "Unit1.Em3.ControlNodes".topTapeFixStage."step".action1[220] := #_w1 AND NOT "Unit1.Em3.ControlNodes".cm.softcam.topTapeAxisY.pos01_load.inPos;
   "Unit1.Em3.ControlNodes".topTapeFixStage."step".transition1[220] := #_w1 AND "Unit1.Em3.ControlNodes".cm.softcam.topTapeAxisY.pos01_load.inPos;
   #statTonTime[220].TON(IN := #_w1 AND "Unit1.Em3.ControlNodes".topTapeFixStage."step".transition1[220],
                         PT := T#500ms);
   IF #statTonTime[220].Q THEN
       "Unit1.Em3.ControlNodes".topTapeFixStage.sequence.status.nextStep := #JOB_2_STEP_30;
   END_IF;
END_REGION

REGION Network 18: Step[230] : Top Tape Fix Stage Bottom Clamp Up
   RUNG wire#powerrail
      { S7_Templates := "SrcType := DInt" } EQ_Contact(in1 := "Unit1.Em3.ControlNodes".topTapeFixStage.sequence.status.currentStep, in2 := #JOB_2_STEP_30)
      Contact( "Unit1.Em3.ControlNodes".topTapeFixStage.sequence.status.seqActive )
      wire#w1
      I_Contact( "Unit1.Em3.ControlNodes".cmTopTapeClampBtmDownUp.monitoring.inWorkPos )
      Coil( "Unit1.Em3.ControlNodes".topTapeFixStage."step".action1[230] )
   END_RUNG
   RUNG wire#w1
      Contact( "Unit1.Em3.ControlNodes".cmTopTapeClampBtmDownUp.monitoring.inWorkPos )
      wire#w2
      Coil( "Unit1.Em3.ControlNodes".topTapeFixStage."step".transition1[230] )
   END_RUNG
   RUNG wire#w1
      Contact( #unitStatus.specialFunctions."Dry Run" )
      Contact( "BA060ZSIPM04.06" )
   END_RUNG wire#w2
   RUNG wire#w1
      Contact( "Unit1.Em3.ControlNodes".topTapeFixStage."step".transition1[230] )
      { S7_Templates := "time_type := Time" } #statTonTime[230].TON(pt := T#500ms, et =>)
      Move(in := #JOB_2_STEP_31, out1 => "Unit1.Em3.ControlNodes".topTapeFixStage.sequence.status.nextStep)
   END_RUNG
   // the same network as SCL:
   #_w1 := ("Unit1.Em3.ControlNodes".topTapeFixStage.sequence.status.currentStep = #JOB_2_STEP_30) AND "Unit1.Em3.ControlNodes".topTapeFixStage.sequence.status.seqActive;
   "Unit1.Em3.ControlNodes".topTapeFixStage."step".action1[230] := #_w1 AND NOT "Unit1.Em3.ControlNodes".cmTopTapeClampBtmDownUp.monitoring.inWorkPos;
   "Unit1.Em3.ControlNodes".topTapeFixStage."step".transition1[230] := #_w1 AND ("Unit1.Em3.ControlNodes".cmTopTapeClampBtmDownUp.monitoring.inWorkPos OR (#unitStatus.specialFunctions."Dry Run" AND "BA060ZSIPM04.06"));
   #statTonTime[230].TON(IN := #_w1 AND "Unit1.Em3.ControlNodes".topTapeFixStage."step".transition1[230],
                         PT := T#500ms);
   IF #statTonTime[230].Q THEN
       "Unit1.Em3.ControlNodes".topTapeFixStage.sequence.status.nextStep := #JOB_2_STEP_31;
   END_IF;
END_REGION

REGION Network 19: Step[231] : Top Tape Fix Stage Left/Center/Right Top Clamp Down
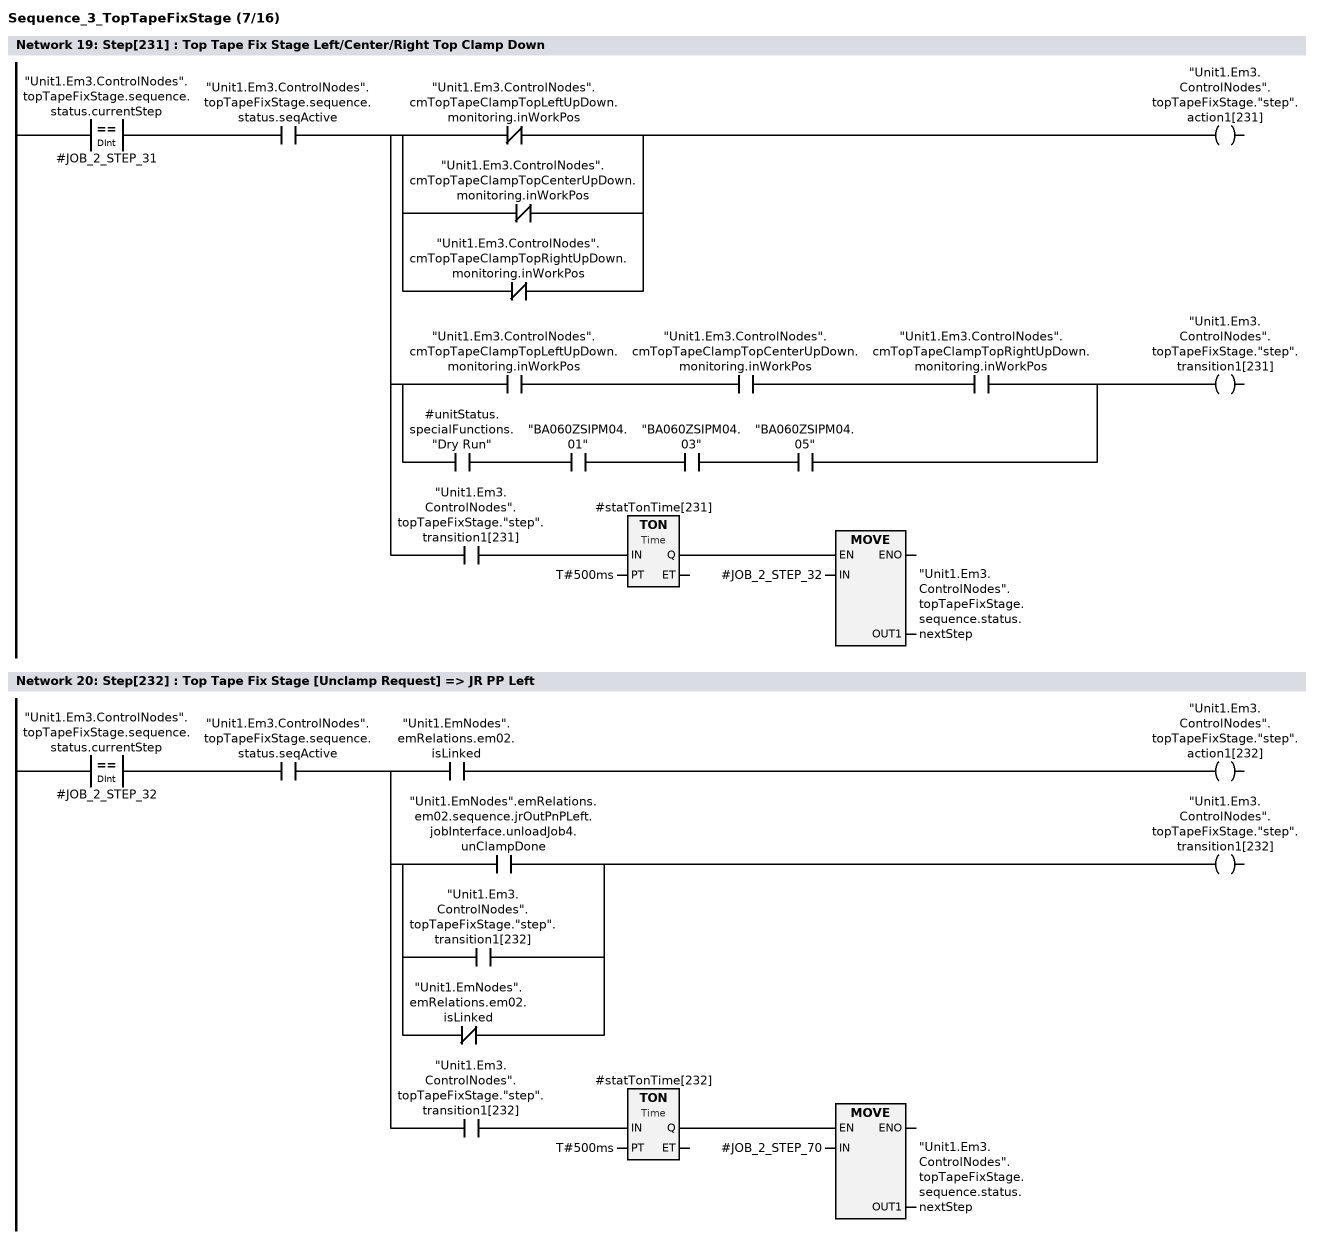
   RUNG wire#powerrail
      { S7_Templates := "SrcType := DInt" } EQ_Contact(in1 := "Unit1.Em3.ControlNodes".topTapeFixStage.sequence.status.currentStep, in2 := #JOB_2_STEP_31)
      Contact( "Unit1.Em3.ControlNodes".topTapeFixStage.sequence.status.seqActive )
      wire#w1
      I_Contact( "Unit1.Em3.ControlNodes".cmTopTapeClampTopLeftUpDown.monitoring.inWorkPos )
      wire#w2
      Coil( "Unit1.Em3.ControlNodes".topTapeFixStage."step".action1[231] )
   END_RUNG
   RUNG wire#w1
      I_Contact( "Unit1.Em3.ControlNodes".cmTopTapeClampTopCenterUpDown.monitoring.inWorkPos )
   END_RUNG wire#w2
   RUNG wire#w1
      I_Contact( "Unit1.Em3.ControlNodes".cmTopTapeClampTopRightUpDown.monitoring.inWorkPos )
   END_RUNG wire#w2
   RUNG wire#w1
      Contact( "Unit1.Em3.ControlNodes".cmTopTapeClampTopLeftUpDown.monitoring.inWorkPos )
      Contact( "Unit1.Em3.ControlNodes".cmTopTapeClampTopCenterUpDown.monitoring.inWorkPos )
      Contact( "Unit1.Em3.ControlNodes".cmTopTapeClampTopRightUpDown.monitoring.inWorkPos )
      wire#w3
      Coil( "Unit1.Em3.ControlNodes".topTapeFixStage."step".transition1[231] )
   END_RUNG
   RUNG wire#w1
      Contact( #unitStatus.specialFunctions."Dry Run" )
      Contact( "BA060ZSIPM04.01" )
      Contact( "BA060ZSIPM04.03" )
      Contact( "BA060ZSIPM04.05" )
   END_RUNG wire#w3
   RUNG wire#w1
      Contact( "Unit1.Em3.ControlNodes".topTapeFixStage."step".transition1[231] )
      { S7_Templates := "time_type := Time" } #statTonTime[231].TON(pt := T#500ms, et =>)
      Move(in := #JOB_2_STEP_32, out1 => "Unit1.Em3.ControlNodes".topTapeFixStage.sequence.status.nextStep)
   END_RUNG
   // the same network as SCL:
   #_w1 := ("Unit1.Em3.ControlNodes".topTapeFixStage.sequence.status.currentStep = #JOB_2_STEP_31) AND "Unit1.Em3.ControlNodes".topTapeFixStage.sequence.status.seqActive;
   "Unit1.Em3.ControlNodes".topTapeFixStage."step".action1[231] := #_w1 AND (NOT "Unit1.Em3.ControlNodes".cmTopTapeClampTopLeftUpDown.monitoring.inWorkPos OR NOT "Unit1.Em3.ControlNodes".cmTopTapeClampTopCenterUpDown.monitoring.inWorkPos OR NOT "Unit1.Em3.ControlNodes".cmTopTapeClampTopRightUpDown.monitoring.inWorkPos);
   "Unit1.Em3.ControlNodes".topTapeFixStage."step".transition1[231] := #_w1 AND (("Unit1.Em3.ControlNodes".cmTopTapeClampTopLeftUpDown.monitoring.inWorkPos AND "Unit1.Em3.ControlNodes".cmTopTapeClampTopCenterUpDown.monitoring.inWorkPos AND "Unit1.Em3.ControlNodes".cmTopTapeClampTopRightUpDown.monitoring.inWorkPos) OR (#unitStatus.specialFunctions."Dry Run" AND "BA060ZSIPM04.01" AND "BA060ZSIPM04.03" AND "BA060ZSIPM04.05"));
   #statTonTime[231].TON(IN := #_w1 AND "Unit1.Em3.ControlNodes".topTapeFixStage."step".transition1[231],
                         PT := T#500ms);
   IF #statTonTime[231].Q THEN
       "Unit1.Em3.ControlNodes".topTapeFixStage.sequence.status.nextStep := #JOB_2_STEP_32;
   END_IF;
END_REGION

REGION Network 20: Step[232] : Top Tape Fix Stage [Unclamp Request] => JR PP Left
   RUNG wire#powerrail
      { S7_Templates := "SrcType := DInt" } EQ_Contact(in1 := "Unit1.Em3.ControlNodes".topTapeFixStage.sequence.status.currentStep, in2 := #JOB_2_STEP_32)
      Contact( "Unit1.Em3.ControlNodes".topTapeFixStage.sequence.status.seqActive )
      wire#w1
      Contact( "Unit1.EmNodes".emRelations.em02.isLinked )
      Coil( "Unit1.Em3.ControlNodes".topTapeFixStage."step".action1[232] )
   END_RUNG
   RUNG wire#w1
      Contact( "Unit1.EmNodes".emRelations.em02.sequence.jrOutPnPLeft.jobInterface.unloadJob4.unClampDone )
      wire#w2
      Coil( "Unit1.Em3.ControlNodes".topTapeFixStage."step".transition1[232] )
   END_RUNG
   RUNG wire#w1
      Contact( "Unit1.Em3.ControlNodes".topTapeFixStage."step".transition1[232] )
   END_RUNG wire#w2
   RUNG wire#w1
      I_Contact( "Unit1.EmNodes".emRelations.em02.isLinked )
   END_RUNG wire#w2
   RUNG wire#w1
      Contact( "Unit1.Em3.ControlNodes".topTapeFixStage."step".transition1[232] )
      { S7_Templates := "time_type := Time" } #statTonTime[232].TON(pt := T#500ms, et =>)
      Move(in := #JOB_2_STEP_70, out1 => "Unit1.Em3.ControlNodes".topTapeFixStage.sequence.status.nextStep)
   END_RUNG
   // the same network as SCL:
   #_w1 := ("Unit1.Em3.ControlNodes".topTapeFixStage.sequence.status.currentStep = #JOB_2_STEP_32) AND "Unit1.Em3.ControlNodes".topTapeFixStage.sequence.status.seqActive;
   "Unit1.Em3.ControlNodes".topTapeFixStage."step".action1[232] := #_w1 AND "Unit1.EmNodes".emRelations.em02.isLinked;
   "Unit1.Em3.ControlNodes".topTapeFixStage."step".transition1[232] := #_w1 AND ("Unit1.EmNodes".emRelations.em02.sequence.jrOutPnPLeft.jobInterface.unloadJob4.unClampDone OR "Unit1.Em3.ControlNodes".topTapeFixStage."step".transition1[232] OR NOT "Unit1.EmNodes".emRelations.em02.isLinked);
   #statTonTime[232].TON(IN := #_w1 AND "Unit1.Em3.ControlNodes".topTapeFixStage."step".transition1[232],
                         PT := T#500ms);
   IF #statTonTime[232].Q THEN
       "Unit1.Em3.ControlNodes".topTapeFixStage.sequence.status.nextStep := #JOB_2_STEP_70;
   END_IF;
END_REGION

REGION Network 21: Step[270] : Spare
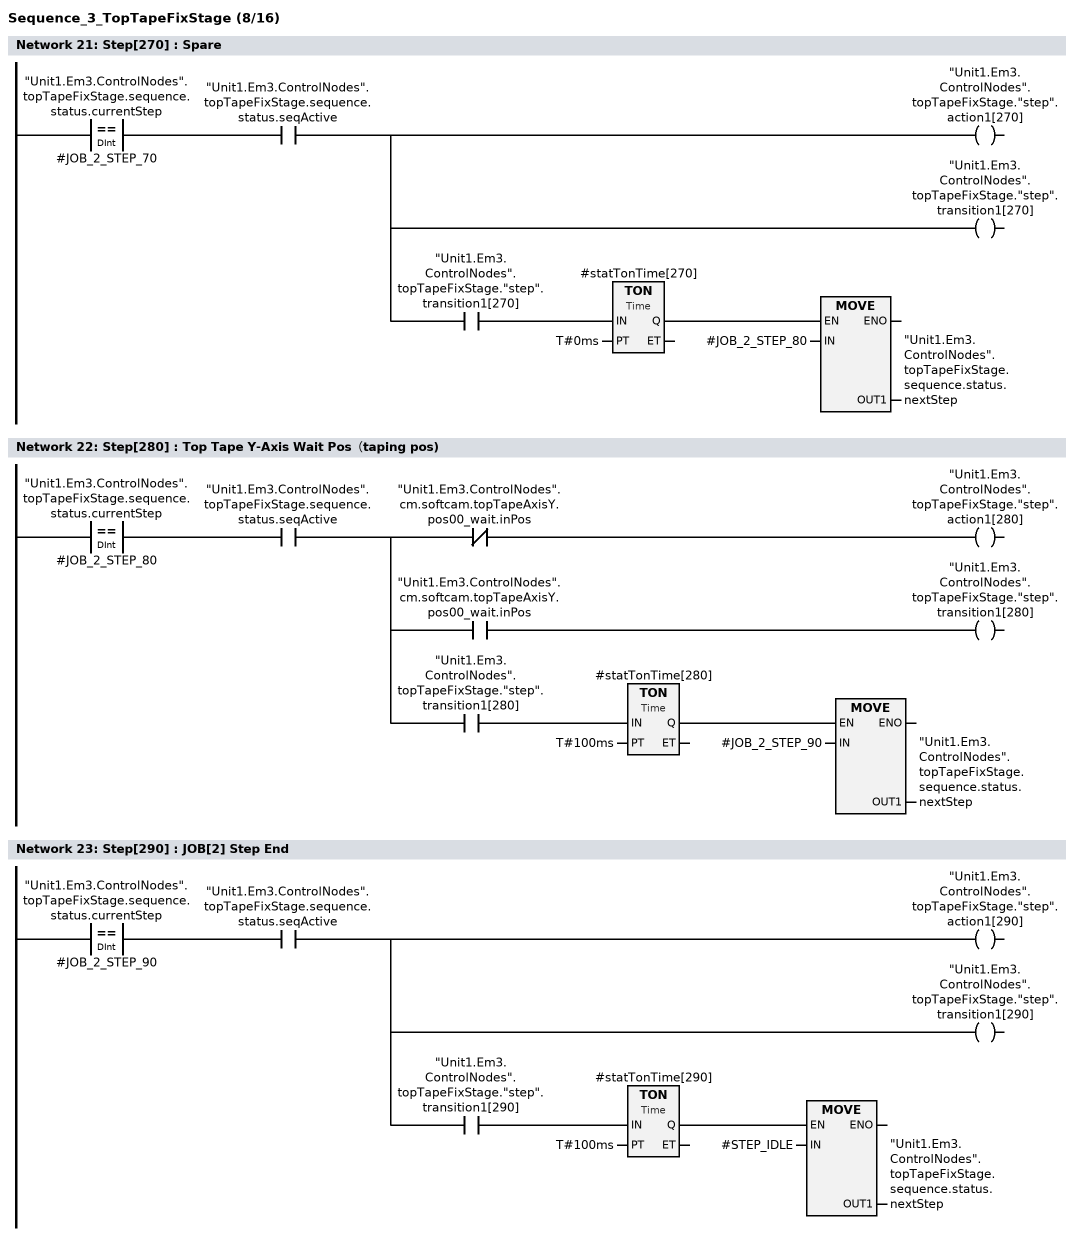
   RUNG wire#powerrail
      { S7_Templates := "SrcType := DInt" } EQ_Contact(in1 := "Unit1.Em3.ControlNodes".topTapeFixStage.sequence.status.currentStep, in2 := #JOB_2_STEP_70)
      Contact( "Unit1.Em3.ControlNodes".topTapeFixStage.sequence.status.seqActive )
      wire#w1
      Coil( "Unit1.Em3.ControlNodes".topTapeFixStage."step".action1[270] )
   END_RUNG
   RUNG wire#w1
      Coil( "Unit1.Em3.ControlNodes".topTapeFixStage."step".transition1[270] )
   END_RUNG
   RUNG wire#w1
      Contact( "Unit1.Em3.ControlNodes".topTapeFixStage."step".transition1[270] )
      { S7_Templates := "time_type := Time" } #statTonTime[270].TON(pt := T#0ms, et =>)
      Move(in := #JOB_2_STEP_80, out1 => "Unit1.Em3.ControlNodes".topTapeFixStage.sequence.status.nextStep)
   END_RUNG
   // the same network as SCL:
   "Unit1.Em3.ControlNodes".topTapeFixStage."step".action1[270] := ("Unit1.Em3.ControlNodes".topTapeFixStage.sequence.status.currentStep = #JOB_2_STEP_70) AND "Unit1.Em3.ControlNodes".topTapeFixStage.sequence.status.seqActive;
   "Unit1.Em3.ControlNodes".topTapeFixStage."step".transition1[270] := ("Unit1.Em3.ControlNodes".topTapeFixStage.sequence.status.currentStep = #JOB_2_STEP_70) AND "Unit1.Em3.ControlNodes".topTapeFixStage.sequence.status.seqActive;
   #statTonTime[270].TON(IN := ("Unit1.Em3.ControlNodes".topTapeFixStage.sequence.status.currentStep = #JOB_2_STEP_70) AND "Unit1.Em3.ControlNodes".topTapeFixStage.sequence.status.seqActive AND "Unit1.Em3.ControlNodes".topTapeFixStage."step".transition1[270],
                         PT := T#0ms);
   IF #statTonTime[270].Q THEN
       "Unit1.Em3.ControlNodes".topTapeFixStage.sequence.status.nextStep := #JOB_2_STEP_80;
   END_IF;
END_REGION

REGION Network 22: Step[280] : Top Tape Y-Axis Wait Pos（taping pos)
   RUNG wire#powerrail
      { S7_Templates := "SrcType := DInt" } EQ_Contact(in1 := "Unit1.Em3.ControlNodes".topTapeFixStage.sequence.status.currentStep, in2 := #JOB_2_STEP_80)
      Contact( "Unit1.Em3.ControlNodes".topTapeFixStage.sequence.status.seqActive )
      wire#w1
      I_Contact( "Unit1.Em3.ControlNodes".cm.softcam.topTapeAxisY.pos00_wait.inPos )
      Coil( "Unit1.Em3.ControlNodes".topTapeFixStage."step".action1[280] )
   END_RUNG
   RUNG wire#w1
      Contact( "Unit1.Em3.ControlNodes".cm.softcam.topTapeAxisY.pos00_wait.inPos )
      Coil( "Unit1.Em3.ControlNodes".topTapeFixStage."step".transition1[280] )
   END_RUNG
   RUNG wire#w1
      Contact( "Unit1.Em3.ControlNodes".topTapeFixStage."step".transition1[280] )
      { S7_Templates := "time_type := Time" } #statTonTime[280].TON(pt := T#100ms, et =>)
      Move(in := #JOB_2_STEP_90, out1 => "Unit1.Em3.ControlNodes".topTapeFixStage.sequence.status.nextStep)
   END_RUNG
   // the same network as SCL:
   #_w1 := ("Unit1.Em3.ControlNodes".topTapeFixStage.sequence.status.currentStep = #JOB_2_STEP_80) AND "Unit1.Em3.ControlNodes".topTapeFixStage.sequence.status.seqActive;
   "Unit1.Em3.ControlNodes".topTapeFixStage."step".action1[280] := #_w1 AND NOT "Unit1.Em3.ControlNodes".cm.softcam.topTapeAxisY.pos00_wait.inPos;
   "Unit1.Em3.ControlNodes".topTapeFixStage."step".transition1[280] := #_w1 AND "Unit1.Em3.ControlNodes".cm.softcam.topTapeAxisY.pos00_wait.inPos;
   #statTonTime[280].TON(IN := #_w1 AND "Unit1.Em3.ControlNodes".topTapeFixStage."step".transition1[280],
                         PT := T#100ms);
   IF #statTonTime[280].Q THEN
       "Unit1.Em3.ControlNodes".topTapeFixStage.sequence.status.nextStep := #JOB_2_STEP_90;
   END_IF;
END_REGION

REGION Network 23: Step[290] : JOB[2] Step End
   RUNG wire#powerrail
      { S7_Templates := "SrcType := DInt" } EQ_Contact(in1 := "Unit1.Em3.ControlNodes".topTapeFixStage.sequence.status.currentStep, in2 := #JOB_2_STEP_90)
      Contact( "Unit1.Em3.ControlNodes".topTapeFixStage.sequence.status.seqActive )
      wire#w1
      Coil( "Unit1.Em3.ControlNodes".topTapeFixStage."step".action1[290] )
   END_RUNG
   RUNG wire#w1
      Coil( "Unit1.Em3.ControlNodes".topTapeFixStage."step".transition1[290] )
   END_RUNG
   RUNG wire#w1
      Contact( "Unit1.Em3.ControlNodes".topTapeFixStage."step".transition1[290] )
      { S7_Templates := "time_type := Time" } #statTonTime[290].TON(pt := T#100ms, et =>)
      Move(in := #STEP_IDLE, out1 => "Unit1.Em3.ControlNodes".topTapeFixStage.sequence.status.nextStep)
   END_RUNG
   // the same network as SCL:
   "Unit1.Em3.ControlNodes".topTapeFixStage."step".action1[290] := ("Unit1.Em3.ControlNodes".topTapeFixStage.sequence.status.currentStep = #JOB_2_STEP_90) AND "Unit1.Em3.ControlNodes".topTapeFixStage.sequence.status.seqActive;
   "Unit1.Em3.ControlNodes".topTapeFixStage."step".transition1[290] := ("Unit1.Em3.ControlNodes".topTapeFixStage.sequence.status.currentStep = #JOB_2_STEP_90) AND "Unit1.Em3.ControlNodes".topTapeFixStage.sequence.status.seqActive;
   #statTonTime[290].TON(IN := ("Unit1.Em3.ControlNodes".topTapeFixStage.sequence.status.currentStep = #JOB_2_STEP_90) AND "Unit1.Em3.ControlNodes".topTapeFixStage.sequence.status.seqActive AND "Unit1.Em3.ControlNodes".topTapeFixStage."step".transition1[290],
                         PT := T#100ms);
   IF #statTonTime[290].Q THEN
       "Unit1.Em3.ControlNodes".topTapeFixStage.sequence.status.nextStep := #STEP_IDLE;
   END_IF;
END_REGION

REGION Network 24: *************** JOB[3] JR TOP TAPING-1=AUTO *************************
END_REGION

REGION Network 25: Step[301] : JOB[3] Conditiion
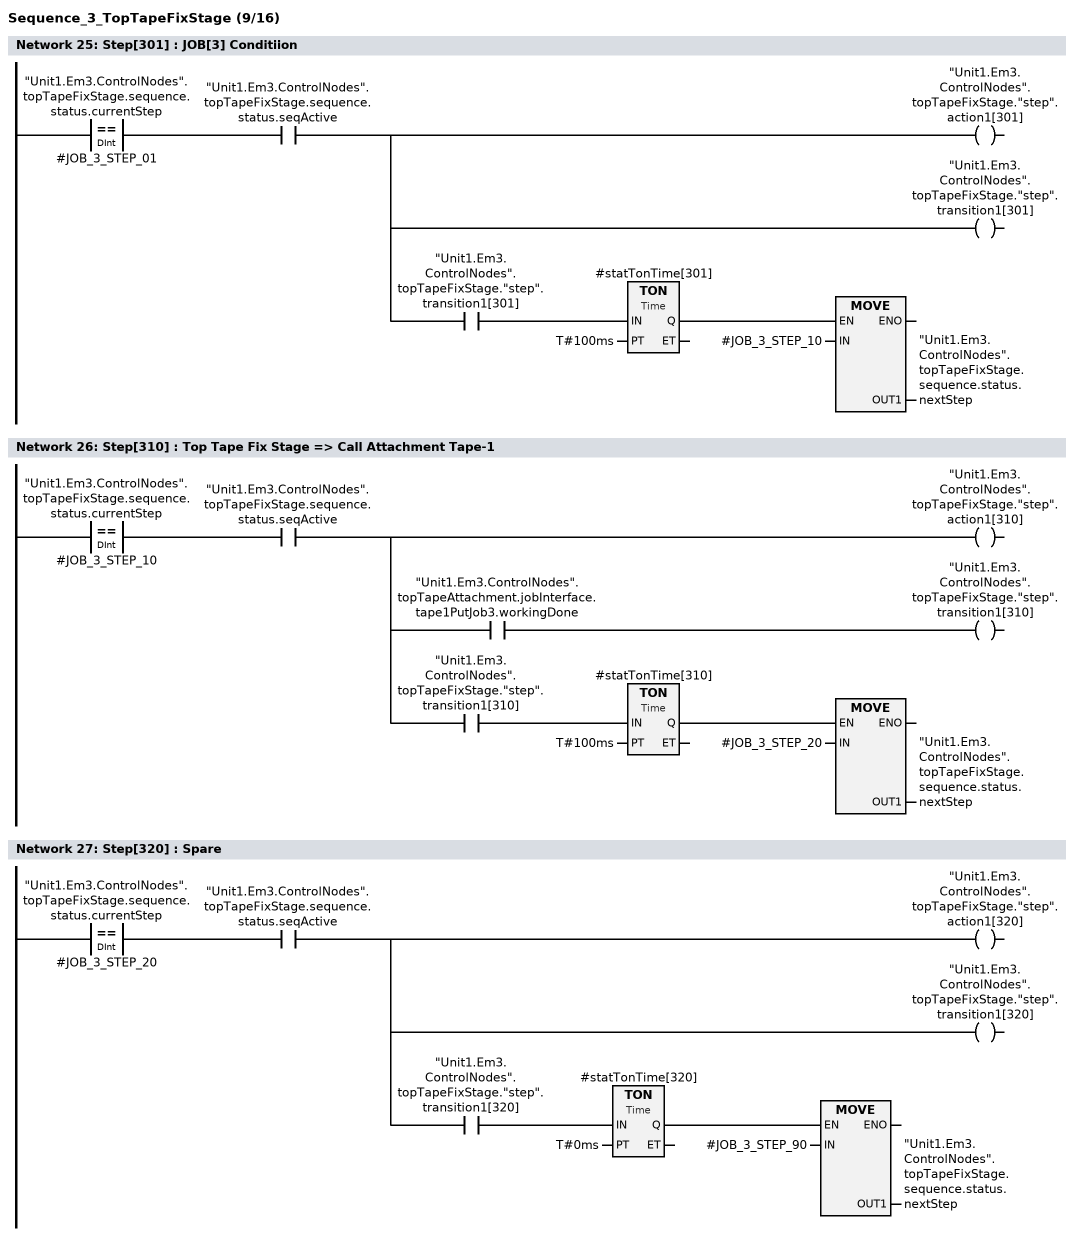
   RUNG wire#powerrail
      { S7_Templates := "SrcType := DInt" } EQ_Contact(in1 := "Unit1.Em3.ControlNodes".topTapeFixStage.sequence.status.currentStep, in2 := #JOB_3_STEP_01)
      Contact( "Unit1.Em3.ControlNodes".topTapeFixStage.sequence.status.seqActive )
      wire#w1
      Coil( "Unit1.Em3.ControlNodes".topTapeFixStage."step".action1[301] )
   END_RUNG
   RUNG wire#w1
      Coil( "Unit1.Em3.ControlNodes".topTapeFixStage."step".transition1[301] )
   END_RUNG
   RUNG wire#w1
      Contact( "Unit1.Em3.ControlNodes".topTapeFixStage."step".transition1[301] )
      { S7_Templates := "time_type := Time" } #statTonTime[301].TON(pt := T#100ms, et =>)
      Move(in := #JOB_3_STEP_10, out1 => "Unit1.Em3.ControlNodes".topTapeFixStage.sequence.status.nextStep)
   END_RUNG
   // the same network as SCL:
   "Unit1.Em3.ControlNodes".topTapeFixStage."step".action1[301] := ("Unit1.Em3.ControlNodes".topTapeFixStage.sequence.status.currentStep = #JOB_3_STEP_01) AND "Unit1.Em3.ControlNodes".topTapeFixStage.sequence.status.seqActive;
   "Unit1.Em3.ControlNodes".topTapeFixStage."step".transition1[301] := ("Unit1.Em3.ControlNodes".topTapeFixStage.sequence.status.currentStep = #JOB_3_STEP_01) AND "Unit1.Em3.ControlNodes".topTapeFixStage.sequence.status.seqActive;
   #statTonTime[301].TON(IN := ("Unit1.Em3.ControlNodes".topTapeFixStage.sequence.status.currentStep = #JOB_3_STEP_01) AND "Unit1.Em3.ControlNodes".topTapeFixStage.sequence.status.seqActive AND "Unit1.Em3.ControlNodes".topTapeFixStage."step".transition1[301],
                         PT := T#100ms);
   IF #statTonTime[301].Q THEN
       "Unit1.Em3.ControlNodes".topTapeFixStage.sequence.status.nextStep := #JOB_3_STEP_10;
   END_IF;
END_REGION

REGION Network 26: Step[310] : Top Tape Fix Stage => Call Attachment Tape-1
   RUNG wire#powerrail
      { S7_Templates := "SrcType := DInt" } EQ_Contact(in1 := "Unit1.Em3.ControlNodes".topTapeFixStage.sequence.status.currentStep, in2 := #JOB_3_STEP_10)
      Contact( "Unit1.Em3.ControlNodes".topTapeFixStage.sequence.status.seqActive )
      wire#w1
      Coil( "Unit1.Em3.ControlNodes".topTapeFixStage."step".action1[310] )
   END_RUNG
   RUNG wire#w1
      Contact( "Unit1.Em3.ControlNodes".topTapeAttachment.jobInterface.tape1PutJob3.workingDone )
      Coil( "Unit1.Em3.ControlNodes".topTapeFixStage."step".transition1[310] )
   END_RUNG
   RUNG wire#w1
      Contact( "Unit1.Em3.ControlNodes".topTapeFixStage."step".transition1[310] )
      { S7_Templates := "time_type := Time" } #statTonTime[310].TON(pt := T#100ms, et =>)
      Move(in := #JOB_3_STEP_20, out1 => "Unit1.Em3.ControlNodes".topTapeFixStage.sequence.status.nextStep)
   END_RUNG
   // the same network as SCL:
   "Unit1.Em3.ControlNodes".topTapeFixStage."step".action1[310] := ("Unit1.Em3.ControlNodes".topTapeFixStage.sequence.status.currentStep = #JOB_3_STEP_10) AND "Unit1.Em3.ControlNodes".topTapeFixStage.sequence.status.seqActive;
   "Unit1.Em3.ControlNodes".topTapeFixStage."step".transition1[310] := ("Unit1.Em3.ControlNodes".topTapeFixStage.sequence.status.currentStep = #JOB_3_STEP_10) AND "Unit1.Em3.ControlNodes".topTapeFixStage.sequence.status.seqActive AND "Unit1.Em3.ControlNodes".topTapeAttachment.jobInterface.tape1PutJob3.workingDone;
   #statTonTime[310].TON(IN := ("Unit1.Em3.ControlNodes".topTapeFixStage.sequence.status.currentStep = #JOB_3_STEP_10) AND "Unit1.Em3.ControlNodes".topTapeFixStage.sequence.status.seqActive AND "Unit1.Em3.ControlNodes".topTapeFixStage."step".transition1[310],
                         PT := T#100ms);
   IF #statTonTime[310].Q THEN
       "Unit1.Em3.ControlNodes".topTapeFixStage.sequence.status.nextStep := #JOB_3_STEP_20;
   END_IF;
END_REGION

REGION Network 27: Step[320] : Spare
   RUNG wire#powerrail
      { S7_Templates := "SrcType := DInt" } EQ_Contact(in1 := "Unit1.Em3.ControlNodes".topTapeFixStage.sequence.status.currentStep, in2 := #JOB_3_STEP_20)
      Contact( "Unit1.Em3.ControlNodes".topTapeFixStage.sequence.status.seqActive )
      wire#w1
      Coil( "Unit1.Em3.ControlNodes".topTapeFixStage."step".action1[320] )
   END_RUNG
   RUNG wire#w1
      Coil( "Unit1.Em3.ControlNodes".topTapeFixStage."step".transition1[320] )
   END_RUNG
   RUNG wire#w1
      Contact( "Unit1.Em3.ControlNodes".topTapeFixStage."step".transition1[320] )
      { S7_Templates := "time_type := Time" } #statTonTime[320].TON(pt := T#0ms, et =>)
      Move(in := #JOB_3_STEP_90, out1 => "Unit1.Em3.ControlNodes".topTapeFixStage.sequence.status.nextStep)
   END_RUNG
   // the same network as SCL:
   "Unit1.Em3.ControlNodes".topTapeFixStage."step".action1[320] := ("Unit1.Em3.ControlNodes".topTapeFixStage.sequence.status.currentStep = #JOB_3_STEP_20) AND "Unit1.Em3.ControlNodes".topTapeFixStage.sequence.status.seqActive;
   "Unit1.Em3.ControlNodes".topTapeFixStage."step".transition1[320] := ("Unit1.Em3.ControlNodes".topTapeFixStage.sequence.status.currentStep = #JOB_3_STEP_20) AND "Unit1.Em3.ControlNodes".topTapeFixStage.sequence.status.seqActive;
   #statTonTime[320].TON(IN := ("Unit1.Em3.ControlNodes".topTapeFixStage.sequence.status.currentStep = #JOB_3_STEP_20) AND "Unit1.Em3.ControlNodes".topTapeFixStage.sequence.status.seqActive AND "Unit1.Em3.ControlNodes".topTapeFixStage."step".transition1[320],
                         PT := T#0ms);
   IF #statTonTime[320].Q THEN
       "Unit1.Em3.ControlNodes".topTapeFixStage.sequence.status.nextStep := #JOB_3_STEP_90;
   END_IF;
END_REGION

REGION Network 28: Step[390] : JOB[3] Step End
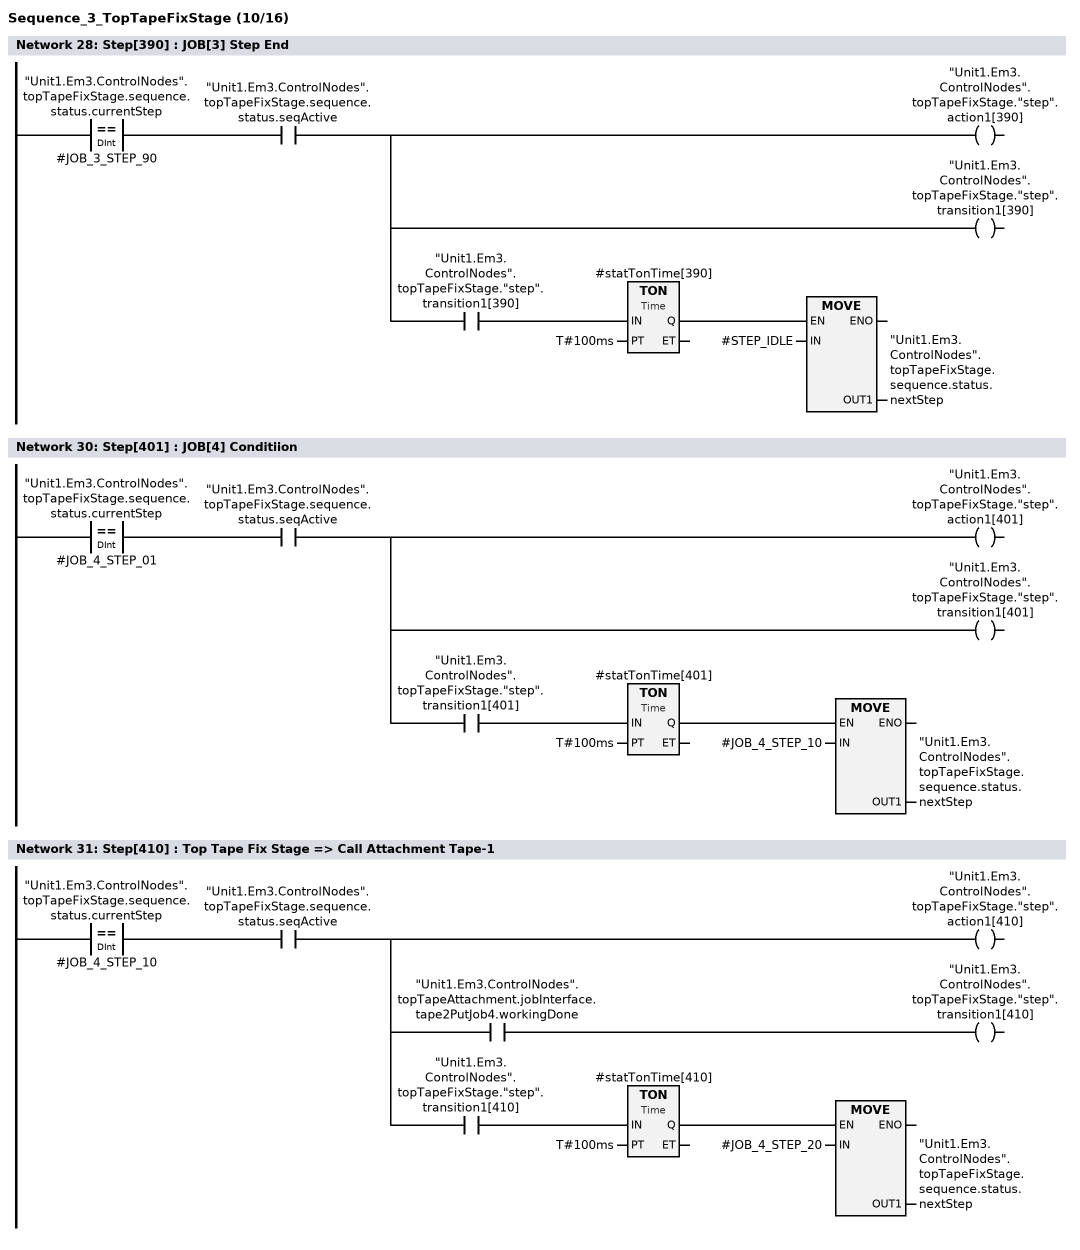
   RUNG wire#powerrail
      { S7_Templates := "SrcType := DInt" } EQ_Contact(in1 := "Unit1.Em3.ControlNodes".topTapeFixStage.sequence.status.currentStep, in2 := #JOB_3_STEP_90)
      Contact( "Unit1.Em3.ControlNodes".topTapeFixStage.sequence.status.seqActive )
      wire#w1
      Coil( "Unit1.Em3.ControlNodes".topTapeFixStage."step".action1[390] )
   END_RUNG
   RUNG wire#w1
      Coil( "Unit1.Em3.ControlNodes".topTapeFixStage."step".transition1[390] )
   END_RUNG
   RUNG wire#w1
      Contact( "Unit1.Em3.ControlNodes".topTapeFixStage."step".transition1[390] )
      { S7_Templates := "time_type := Time" } #statTonTime[390].TON(pt := T#100ms, et =>)
      Move(in := #STEP_IDLE, out1 => "Unit1.Em3.ControlNodes".topTapeFixStage.sequence.status.nextStep)
   END_RUNG
   // the same network as SCL:
   "Unit1.Em3.ControlNodes".topTapeFixStage."step".action1[390] := ("Unit1.Em3.ControlNodes".topTapeFixStage.sequence.status.currentStep = #JOB_3_STEP_90) AND "Unit1.Em3.ControlNodes".topTapeFixStage.sequence.status.seqActive;
   "Unit1.Em3.ControlNodes".topTapeFixStage."step".transition1[390] := ("Unit1.Em3.ControlNodes".topTapeFixStage.sequence.status.currentStep = #JOB_3_STEP_90) AND "Unit1.Em3.ControlNodes".topTapeFixStage.sequence.status.seqActive;
   #statTonTime[390].TON(IN := ("Unit1.Em3.ControlNodes".topTapeFixStage.sequence.status.currentStep = #JOB_3_STEP_90) AND "Unit1.Em3.ControlNodes".topTapeFixStage.sequence.status.seqActive AND "Unit1.Em3.ControlNodes".topTapeFixStage."step".transition1[390],
                         PT := T#100ms);
   IF #statTonTime[390].Q THEN
       "Unit1.Em3.ControlNodes".topTapeFixStage.sequence.status.nextStep := #STEP_IDLE;
   END_IF;
END_REGION

REGION Network 29: *************** JOB[4] JR TOP TAPING-2=AUTO *************************
END_REGION

REGION Network 30: Step[401] : JOB[4] Conditiion
   RUNG wire#powerrail
      { S7_Templates := "SrcType := DInt" } EQ_Contact(in1 := "Unit1.Em3.ControlNodes".topTapeFixStage.sequence.status.currentStep, in2 := #JOB_4_STEP_01)
      Contact( "Unit1.Em3.ControlNodes".topTapeFixStage.sequence.status.seqActive )
      wire#w1
      Coil( "Unit1.Em3.ControlNodes".topTapeFixStage."step".action1[401] )
   END_RUNG
   RUNG wire#w1
      Coil( "Unit1.Em3.ControlNodes".topTapeFixStage."step".transition1[401] )
   END_RUNG
   RUNG wire#w1
      Contact( "Unit1.Em3.ControlNodes".topTapeFixStage."step".transition1[401] )
      { S7_Templates := "time_type := Time" } #statTonTime[401].TON(pt := T#100ms, et =>)
      Move(in := #JOB_4_STEP_10, out1 => "Unit1.Em3.ControlNodes".topTapeFixStage.sequence.status.nextStep)
   END_RUNG
   // the same network as SCL:
   "Unit1.Em3.ControlNodes".topTapeFixStage."step".action1[401] := ("Unit1.Em3.ControlNodes".topTapeFixStage.sequence.status.currentStep = #JOB_4_STEP_01) AND "Unit1.Em3.ControlNodes".topTapeFixStage.sequence.status.seqActive;
   "Unit1.Em3.ControlNodes".topTapeFixStage."step".transition1[401] := ("Unit1.Em3.ControlNodes".topTapeFixStage.sequence.status.currentStep = #JOB_4_STEP_01) AND "Unit1.Em3.ControlNodes".topTapeFixStage.sequence.status.seqActive;
   #statTonTime[401].TON(IN := ("Unit1.Em3.ControlNodes".topTapeFixStage.sequence.status.currentStep = #JOB_4_STEP_01) AND "Unit1.Em3.ControlNodes".topTapeFixStage.sequence.status.seqActive AND "Unit1.Em3.ControlNodes".topTapeFixStage."step".transition1[401],
                         PT := T#100ms);
   IF #statTonTime[401].Q THEN
       "Unit1.Em3.ControlNodes".topTapeFixStage.sequence.status.nextStep := #JOB_4_STEP_10;
   END_IF;
END_REGION

REGION Network 31: Step[410] : Top Tape Fix Stage => Call Attachment Tape-1
   RUNG wire#powerrail
      { S7_Templates := "SrcType := DInt" } EQ_Contact(in1 := "Unit1.Em3.ControlNodes".topTapeFixStage.sequence.status.currentStep, in2 := #JOB_4_STEP_10)
      Contact( "Unit1.Em3.ControlNodes".topTapeFixStage.sequence.status.seqActive )
      wire#w1
      Coil( "Unit1.Em3.ControlNodes".topTapeFixStage."step".action1[410] )
   END_RUNG
   RUNG wire#w1
      Contact( "Unit1.Em3.ControlNodes".topTapeAttachment.jobInterface.tape2PutJob4.workingDone )
      Coil( "Unit1.Em3.ControlNodes".topTapeFixStage."step".transition1[410] )
   END_RUNG
   RUNG wire#w1
      Contact( "Unit1.Em3.ControlNodes".topTapeFixStage."step".transition1[410] )
      { S7_Templates := "time_type := Time" } #statTonTime[410].TON(pt := T#100ms, et =>)
      Move(in := #JOB_4_STEP_20, out1 => "Unit1.Em3.ControlNodes".topTapeFixStage.sequence.status.nextStep)
   END_RUNG
   // the same network as SCL:
   "Unit1.Em3.ControlNodes".topTapeFixStage."step".action1[410] := ("Unit1.Em3.ControlNodes".topTapeFixStage.sequence.status.currentStep = #JOB_4_STEP_10) AND "Unit1.Em3.ControlNodes".topTapeFixStage.sequence.status.seqActive;
   "Unit1.Em3.ControlNodes".topTapeFixStage."step".transition1[410] := ("Unit1.Em3.ControlNodes".topTapeFixStage.sequence.status.currentStep = #JOB_4_STEP_10) AND "Unit1.Em3.ControlNodes".topTapeFixStage.sequence.status.seqActive AND "Unit1.Em3.ControlNodes".topTapeAttachment.jobInterface.tape2PutJob4.workingDone;
   #statTonTime[410].TON(IN := ("Unit1.Em3.ControlNodes".topTapeFixStage.sequence.status.currentStep = #JOB_4_STEP_10) AND "Unit1.Em3.ControlNodes".topTapeFixStage.sequence.status.seqActive AND "Unit1.Em3.ControlNodes".topTapeFixStage."step".transition1[410],
                         PT := T#100ms);
   IF #statTonTime[410].Q THEN
       "Unit1.Em3.ControlNodes".topTapeFixStage.sequence.status.nextStep := #JOB_4_STEP_20;
   END_IF;
END_REGION

REGION Network 32: Step[420] : Spare
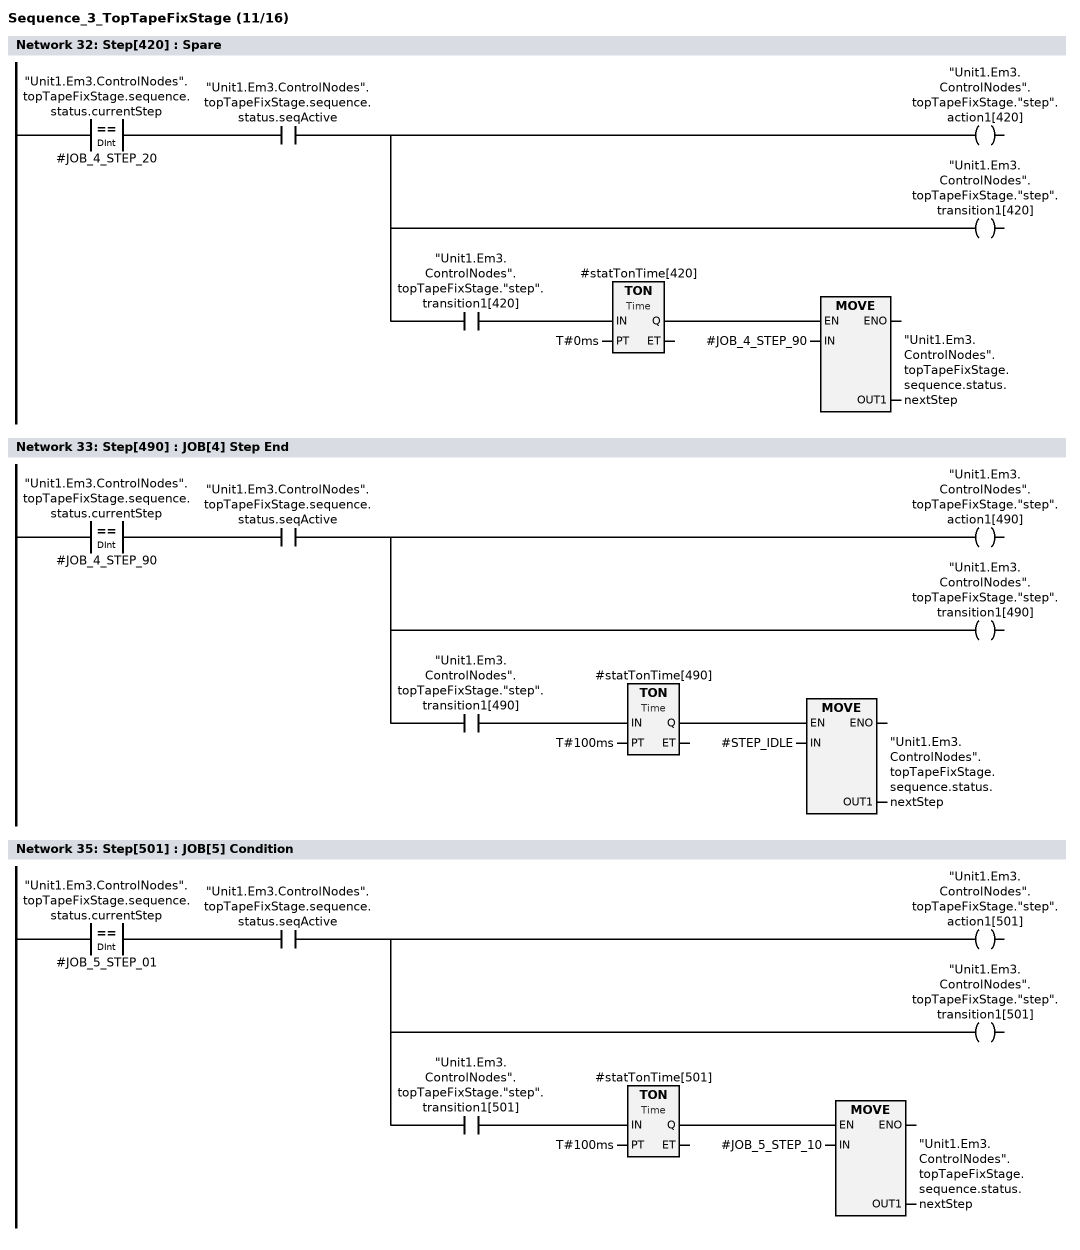
   RUNG wire#powerrail
      { S7_Templates := "SrcType := DInt" } EQ_Contact(in1 := "Unit1.Em3.ControlNodes".topTapeFixStage.sequence.status.currentStep, in2 := #JOB_4_STEP_20)
      Contact( "Unit1.Em3.ControlNodes".topTapeFixStage.sequence.status.seqActive )
      wire#w1
      Coil( "Unit1.Em3.ControlNodes".topTapeFixStage."step".action1[420] )
   END_RUNG
   RUNG wire#w1
      Coil( "Unit1.Em3.ControlNodes".topTapeFixStage."step".transition1[420] )
   END_RUNG
   RUNG wire#w1
      Contact( "Unit1.Em3.ControlNodes".topTapeFixStage."step".transition1[420] )
      { S7_Templates := "time_type := Time" } #statTonTime[420].TON(pt := T#0ms, et =>)
      Move(in := #JOB_4_STEP_90, out1 => "Unit1.Em3.ControlNodes".topTapeFixStage.sequence.status.nextStep)
   END_RUNG
   // the same network as SCL:
   "Unit1.Em3.ControlNodes".topTapeFixStage."step".action1[420] := ("Unit1.Em3.ControlNodes".topTapeFixStage.sequence.status.currentStep = #JOB_4_STEP_20) AND "Unit1.Em3.ControlNodes".topTapeFixStage.sequence.status.seqActive;
   "Unit1.Em3.ControlNodes".topTapeFixStage."step".transition1[420] := ("Unit1.Em3.ControlNodes".topTapeFixStage.sequence.status.currentStep = #JOB_4_STEP_20) AND "Unit1.Em3.ControlNodes".topTapeFixStage.sequence.status.seqActive;
   #statTonTime[420].TON(IN := ("Unit1.Em3.ControlNodes".topTapeFixStage.sequence.status.currentStep = #JOB_4_STEP_20) AND "Unit1.Em3.ControlNodes".topTapeFixStage.sequence.status.seqActive AND "Unit1.Em3.ControlNodes".topTapeFixStage."step".transition1[420],
                         PT := T#0ms);
   IF #statTonTime[420].Q THEN
       "Unit1.Em3.ControlNodes".topTapeFixStage.sequence.status.nextStep := #JOB_4_STEP_90;
   END_IF;
END_REGION

REGION Network 33: Step[490] : JOB[4] Step End
   RUNG wire#powerrail
      { S7_Templates := "SrcType := DInt" } EQ_Contact(in1 := "Unit1.Em3.ControlNodes".topTapeFixStage.sequence.status.currentStep, in2 := #JOB_4_STEP_90)
      Contact( "Unit1.Em3.ControlNodes".topTapeFixStage.sequence.status.seqActive )
      wire#w1
      Coil( "Unit1.Em3.ControlNodes".topTapeFixStage."step".action1[490] )
   END_RUNG
   RUNG wire#w1
      Coil( "Unit1.Em3.ControlNodes".topTapeFixStage."step".transition1[490] )
   END_RUNG
   RUNG wire#w1
      Contact( "Unit1.Em3.ControlNodes".topTapeFixStage."step".transition1[490] )
      { S7_Templates := "time_type := Time" } #statTonTime[490].TON(pt := T#100ms, et =>)
      Move(in := #STEP_IDLE, out1 => "Unit1.Em3.ControlNodes".topTapeFixStage.sequence.status.nextStep)
   END_RUNG
   // the same network as SCL:
   "Unit1.Em3.ControlNodes".topTapeFixStage."step".action1[490] := ("Unit1.Em3.ControlNodes".topTapeFixStage.sequence.status.currentStep = #JOB_4_STEP_90) AND "Unit1.Em3.ControlNodes".topTapeFixStage.sequence.status.seqActive;
   "Unit1.Em3.ControlNodes".topTapeFixStage."step".transition1[490] := ("Unit1.Em3.ControlNodes".topTapeFixStage.sequence.status.currentStep = #JOB_4_STEP_90) AND "Unit1.Em3.ControlNodes".topTapeFixStage.sequence.status.seqActive;
   #statTonTime[490].TON(IN := ("Unit1.Em3.ControlNodes".topTapeFixStage.sequence.status.currentStep = #JOB_4_STEP_90) AND "Unit1.Em3.ControlNodes".topTapeFixStage.sequence.status.seqActive AND "Unit1.Em3.ControlNodes".topTapeFixStage."step".transition1[490],
                         PT := T#100ms);
   IF #statTonTime[490].Q THEN
       "Unit1.Em3.ControlNodes".topTapeFixStage.sequence.status.nextStep := #STEP_IDLE;
   END_IF;
END_REGION

REGION Network 34: *************** JOB[5] JR PUT=AUTO *************************
END_REGION

REGION Network 35: Step[501] : JOB[5] Condition
   RUNG wire#powerrail
      { S7_Templates := "SrcType := DInt" } EQ_Contact(in1 := "Unit1.Em3.ControlNodes".topTapeFixStage.sequence.status.currentStep, in2 := #JOB_5_STEP_01)
      Contact( "Unit1.Em3.ControlNodes".topTapeFixStage.sequence.status.seqActive )
      wire#w1
      Coil( "Unit1.Em3.ControlNodes".topTapeFixStage."step".action1[501] )
   END_RUNG
   RUNG wire#w1
      Coil( "Unit1.Em3.ControlNodes".topTapeFixStage."step".transition1[501] )
   END_RUNG
   RUNG wire#w1
      Contact( "Unit1.Em3.ControlNodes".topTapeFixStage."step".transition1[501] )
      { S7_Templates := "time_type := Time" } #statTonTime[501].TON(pt := T#100ms, et =>)
      Move(in := #JOB_5_STEP_10, out1 => "Unit1.Em3.ControlNodes".topTapeFixStage.sequence.status.nextStep)
   END_RUNG
   // the same network as SCL:
   "Unit1.Em3.ControlNodes".topTapeFixStage."step".action1[501] := ("Unit1.Em3.ControlNodes".topTapeFixStage.sequence.status.currentStep = #JOB_5_STEP_01) AND "Unit1.Em3.ControlNodes".topTapeFixStage.sequence.status.seqActive;
   "Unit1.Em3.ControlNodes".topTapeFixStage."step".transition1[501] := ("Unit1.Em3.ControlNodes".topTapeFixStage.sequence.status.currentStep = #JOB_5_STEP_01) AND "Unit1.Em3.ControlNodes".topTapeFixStage.sequence.status.seqActive;
   #statTonTime[501].TON(IN := ("Unit1.Em3.ControlNodes".topTapeFixStage.sequence.status.currentStep = #JOB_5_STEP_01) AND "Unit1.Em3.ControlNodes".topTapeFixStage.sequence.status.seqActive AND "Unit1.Em3.ControlNodes".topTapeFixStage."step".transition1[501],
                         PT := T#100ms);
   IF #statTonTime[501].Q THEN
       "Unit1.Em3.ControlNodes".topTapeFixStage.sequence.status.nextStep := #JOB_5_STEP_10;
   END_IF;
END_REGION

REGION Network 36: Step[510] : Top Tape Fix Stage [Unloading Request] => JR PP Right
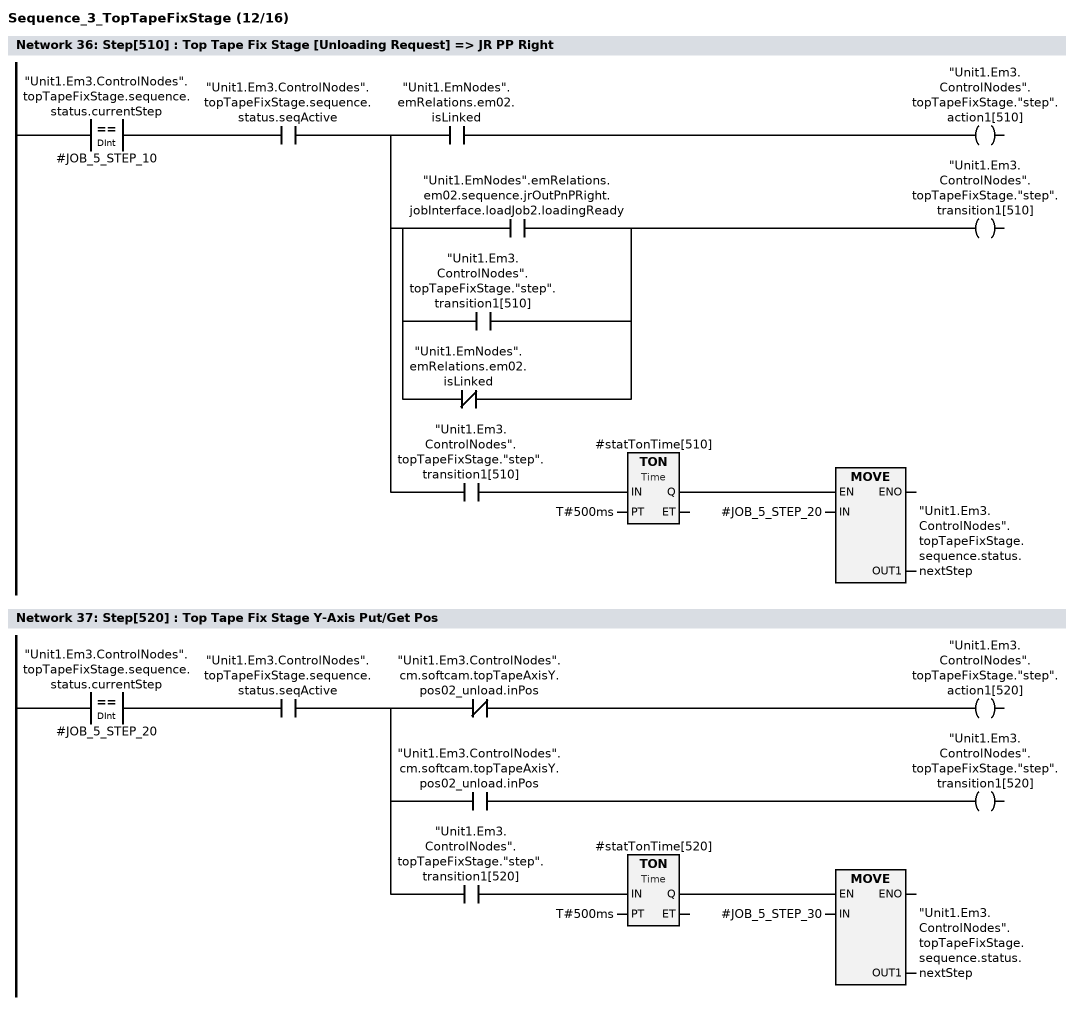
   RUNG wire#powerrail
      { S7_Templates := "SrcType := DInt" } EQ_Contact(in1 := "Unit1.Em3.ControlNodes".topTapeFixStage.sequence.status.currentStep, in2 := #JOB_5_STEP_10)
      Contact( "Unit1.Em3.ControlNodes".topTapeFixStage.sequence.status.seqActive )
      wire#w1
      Contact( "Unit1.EmNodes".emRelations.em02.isLinked )
      Coil( "Unit1.Em3.ControlNodes".topTapeFixStage."step".action1[510] )
   END_RUNG
   RUNG wire#w1
      Contact( "Unit1.EmNodes".emRelations.em02.sequence.jrOutPnPRight.jobInterface.loadJob2.loadingReady )
      wire#w2
      Coil( "Unit1.Em3.ControlNodes".topTapeFixStage."step".transition1[510] )
   END_RUNG
   RUNG wire#w1
      Contact( "Unit1.Em3.ControlNodes".topTapeFixStage."step".transition1[510] )
   END_RUNG wire#w2
   RUNG wire#w1
      I_Contact( "Unit1.EmNodes".emRelations.em02.isLinked )
   END_RUNG wire#w2
   RUNG wire#w1
      Contact( "Unit1.Em3.ControlNodes".topTapeFixStage."step".transition1[510] )
      { S7_Templates := "time_type := Time" } #statTonTime[510].TON(pt := T#500ms, et =>)
      Move(in := #JOB_5_STEP_20, out1 => "Unit1.Em3.ControlNodes".topTapeFixStage.sequence.status.nextStep)
   END_RUNG
   // the same network as SCL:
   #_w1 := ("Unit1.Em3.ControlNodes".topTapeFixStage.sequence.status.currentStep = #JOB_5_STEP_10) AND "Unit1.Em3.ControlNodes".topTapeFixStage.sequence.status.seqActive;
   "Unit1.Em3.ControlNodes".topTapeFixStage."step".action1[510] := #_w1 AND "Unit1.EmNodes".emRelations.em02.isLinked;
   "Unit1.Em3.ControlNodes".topTapeFixStage."step".transition1[510] := #_w1 AND ("Unit1.EmNodes".emRelations.em02.sequence.jrOutPnPRight.jobInterface.loadJob2.loadingReady OR "Unit1.Em3.ControlNodes".topTapeFixStage."step".transition1[510] OR NOT "Unit1.EmNodes".emRelations.em02.isLinked);
   #statTonTime[510].TON(IN := #_w1 AND "Unit1.Em3.ControlNodes".topTapeFixStage."step".transition1[510],
                         PT := T#500ms);
   IF #statTonTime[510].Q THEN
       "Unit1.Em3.ControlNodes".topTapeFixStage.sequence.status.nextStep := #JOB_5_STEP_20;
   END_IF;
END_REGION

REGION Network 37: Step[520] : Top Tape Fix Stage Y-Axis Put/Get Pos
   RUNG wire#powerrail
      { S7_Templates := "SrcType := DInt" } EQ_Contact(in1 := "Unit1.Em3.ControlNodes".topTapeFixStage.sequence.status.currentStep, in2 := #JOB_5_STEP_20)
      Contact( "Unit1.Em3.ControlNodes".topTapeFixStage.sequence.status.seqActive )
      wire#w1
      I_Contact( "Unit1.Em3.ControlNodes".cm.softcam.topTapeAxisY.pos02_unload.inPos )
      Coil( "Unit1.Em3.ControlNodes".topTapeFixStage."step".action1[520] )
   END_RUNG
   RUNG wire#w1
      Contact( "Unit1.Em3.ControlNodes".cm.softcam.topTapeAxisY.pos02_unload.inPos )
      Coil( "Unit1.Em3.ControlNodes".topTapeFixStage."step".transition1[520] )
   END_RUNG
   RUNG wire#w1
      Contact( "Unit1.Em3.ControlNodes".topTapeFixStage."step".transition1[520] )
      { S7_Templates := "time_type := Time" } #statTonTime[520].TON(pt := T#500ms, et =>)
      Move(in := #JOB_5_STEP_30, out1 => "Unit1.Em3.ControlNodes".topTapeFixStage.sequence.status.nextStep)
   END_RUNG
   // the same network as SCL:
   #_w1 := ("Unit1.Em3.ControlNodes".topTapeFixStage.sequence.status.currentStep = #JOB_5_STEP_20) AND "Unit1.Em3.ControlNodes".topTapeFixStage.sequence.status.seqActive;
   "Unit1.Em3.ControlNodes".topTapeFixStage."step".action1[520] := #_w1 AND NOT "Unit1.Em3.ControlNodes".cm.softcam.topTapeAxisY.pos02_unload.inPos;
   "Unit1.Em3.ControlNodes".topTapeFixStage."step".transition1[520] := #_w1 AND "Unit1.Em3.ControlNodes".cm.softcam.topTapeAxisY.pos02_unload.inPos;
   #statTonTime[520].TON(IN := #_w1 AND "Unit1.Em3.ControlNodes".topTapeFixStage."step".transition1[520],
                         PT := T#500ms);
   IF #statTonTime[520].Q THEN
       "Unit1.Em3.ControlNodes".topTapeFixStage.sequence.status.nextStep := #JOB_5_STEP_30;
   END_IF;
END_REGION

REGION Network 38: Step[530] : Top Tape Fix Stage [Clamp Request] => JR PP Right
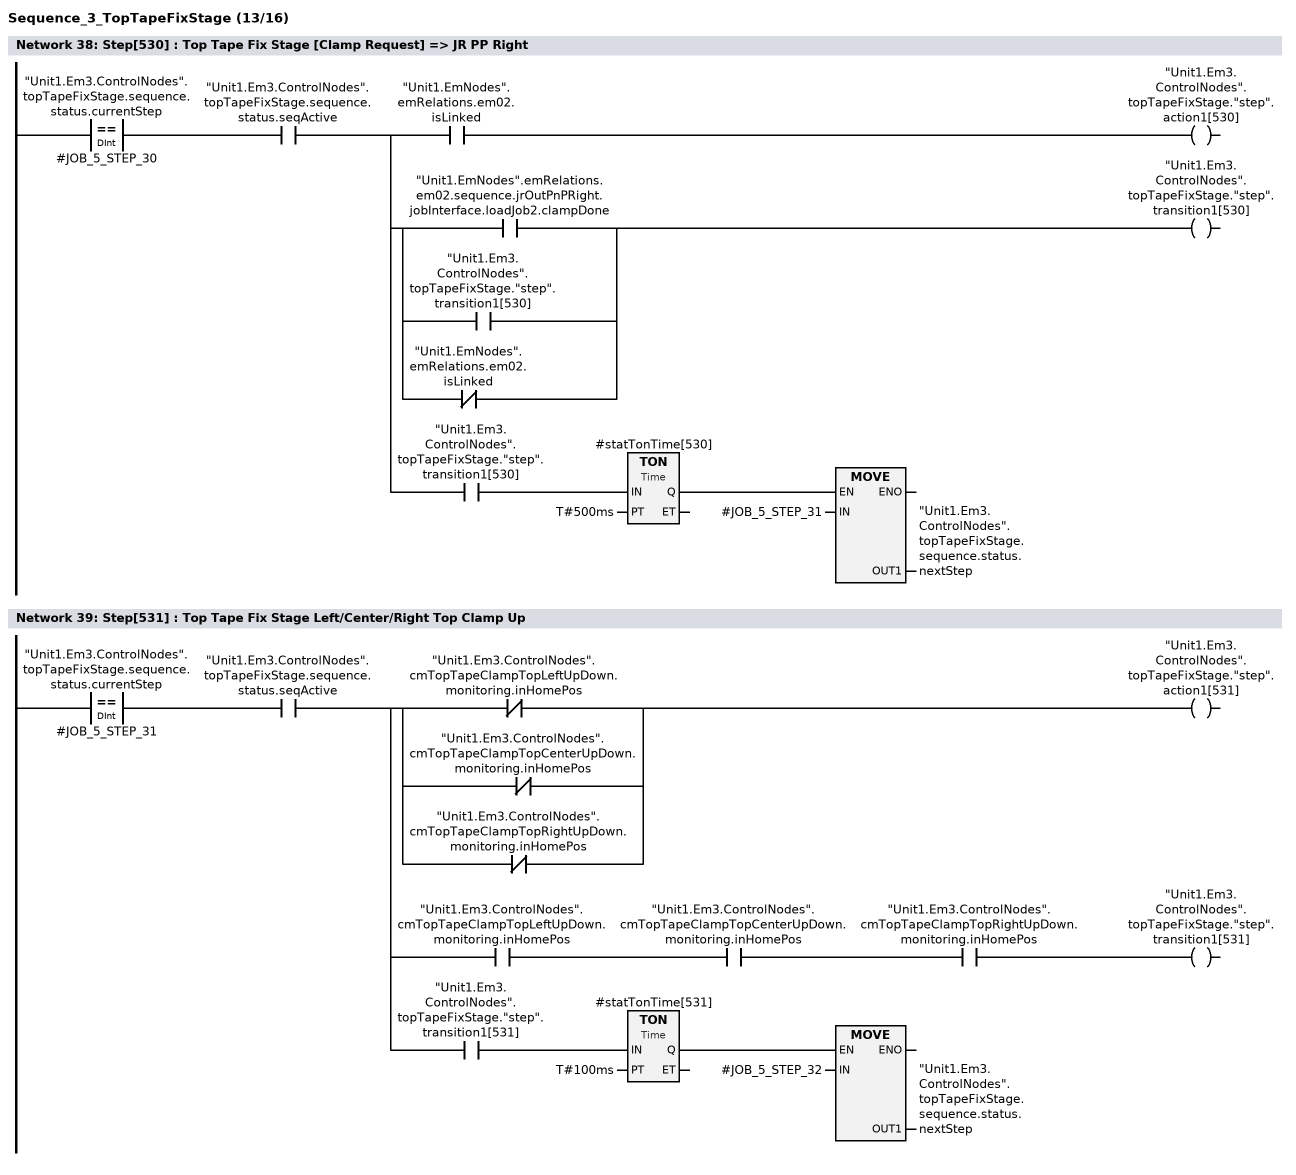
   RUNG wire#powerrail
      { S7_Templates := "SrcType := DInt" } EQ_Contact(in1 := "Unit1.Em3.ControlNodes".topTapeFixStage.sequence.status.currentStep, in2 := #JOB_5_STEP_30)
      Contact( "Unit1.Em3.ControlNodes".topTapeFixStage.sequence.status.seqActive )
      wire#w1
      Contact( "Unit1.EmNodes".emRelations.em02.isLinked )
      Coil( "Unit1.Em3.ControlNodes".topTapeFixStage."step".action1[530] )
   END_RUNG
   RUNG wire#w1
      Contact( "Unit1.EmNodes".emRelations.em02.sequence.jrOutPnPRight.jobInterface.loadJob2.clampDone )
      wire#w2
      Coil( "Unit1.Em3.ControlNodes".topTapeFixStage."step".transition1[530] )
   END_RUNG
   RUNG wire#w1
      Contact( "Unit1.Em3.ControlNodes".topTapeFixStage."step".transition1[530] )
   END_RUNG wire#w2
   RUNG wire#w1
      I_Contact( "Unit1.EmNodes".emRelations.em02.isLinked )
   END_RUNG wire#w2
   RUNG wire#w1
      Contact( "Unit1.Em3.ControlNodes".topTapeFixStage."step".transition1[530] )
      { S7_Templates := "time_type := Time" } #statTonTime[530].TON(pt := T#500ms, et =>)
      Move(in := #JOB_5_STEP_31, out1 => "Unit1.Em3.ControlNodes".topTapeFixStage.sequence.status.nextStep)
   END_RUNG
   // the same network as SCL:
   #_w1 := ("Unit1.Em3.ControlNodes".topTapeFixStage.sequence.status.currentStep = #JOB_5_STEP_30) AND "Unit1.Em3.ControlNodes".topTapeFixStage.sequence.status.seqActive;
   "Unit1.Em3.ControlNodes".topTapeFixStage."step".action1[530] := #_w1 AND "Unit1.EmNodes".emRelations.em02.isLinked;
   "Unit1.Em3.ControlNodes".topTapeFixStage."step".transition1[530] := #_w1 AND ("Unit1.EmNodes".emRelations.em02.sequence.jrOutPnPRight.jobInterface.loadJob2.clampDone OR "Unit1.Em3.ControlNodes".topTapeFixStage."step".transition1[530] OR NOT "Unit1.EmNodes".emRelations.em02.isLinked);
   #statTonTime[530].TON(IN := #_w1 AND "Unit1.Em3.ControlNodes".topTapeFixStage."step".transition1[530],
                         PT := T#500ms);
   IF #statTonTime[530].Q THEN
       "Unit1.Em3.ControlNodes".topTapeFixStage.sequence.status.nextStep := #JOB_5_STEP_31;
   END_IF;
END_REGION

REGION Network 39: Step[531] : Top Tape Fix Stage Left/Center/Right Top Clamp Up
   RUNG wire#powerrail
      { S7_Templates := "SrcType := DInt" } EQ_Contact(in1 := "Unit1.Em3.ControlNodes".topTapeFixStage.sequence.status.currentStep, in2 := #JOB_5_STEP_31)
      Contact( "Unit1.Em3.ControlNodes".topTapeFixStage.sequence.status.seqActive )
      wire#w1
      I_Contact( "Unit1.Em3.ControlNodes".cmTopTapeClampTopLeftUpDown.monitoring.inHomePos )
      wire#w2
      Coil( "Unit1.Em3.ControlNodes".topTapeFixStage."step".action1[531] )
   END_RUNG
   RUNG wire#w1
      I_Contact( "Unit1.Em3.ControlNodes".cmTopTapeClampTopCenterUpDown.monitoring.inHomePos )
   END_RUNG wire#w2
   RUNG wire#w1
      I_Contact( "Unit1.Em3.ControlNodes".cmTopTapeClampTopRightUpDown.monitoring.inHomePos )
   END_RUNG wire#w2
   RUNG wire#w1
      Contact( "Unit1.Em3.ControlNodes".cmTopTapeClampTopLeftUpDown.monitoring.inHomePos )
      Contact( "Unit1.Em3.ControlNodes".cmTopTapeClampTopCenterUpDown.monitoring.inHomePos )
      Contact( "Unit1.Em3.ControlNodes".cmTopTapeClampTopRightUpDown.monitoring.inHomePos )
      Coil( "Unit1.Em3.ControlNodes".topTapeFixStage."step".transition1[531] )
   END_RUNG
   RUNG wire#w1
      Contact( "Unit1.Em3.ControlNodes".topTapeFixStage."step".transition1[531] )
      { S7_Templates := "time_type := Time" } #statTonTime[531].TON(pt := T#100ms, et =>)
      Move(in := #JOB_5_STEP_32, out1 => "Unit1.Em3.ControlNodes".topTapeFixStage.sequence.status.nextStep)
   END_RUNG
   // the same network as SCL:
   #_w1 := ("Unit1.Em3.ControlNodes".topTapeFixStage.sequence.status.currentStep = #JOB_5_STEP_31) AND "Unit1.Em3.ControlNodes".topTapeFixStage.sequence.status.seqActive;
   "Unit1.Em3.ControlNodes".topTapeFixStage."step".action1[531] := #_w1 AND (NOT "Unit1.Em3.ControlNodes".cmTopTapeClampTopLeftUpDown.monitoring.inHomePos OR NOT "Unit1.Em3.ControlNodes".cmTopTapeClampTopCenterUpDown.monitoring.inHomePos OR NOT "Unit1.Em3.ControlNodes".cmTopTapeClampTopRightUpDown.monitoring.inHomePos);
   "Unit1.Em3.ControlNodes".topTapeFixStage."step".transition1[531] := #_w1 AND "Unit1.Em3.ControlNodes".cmTopTapeClampTopLeftUpDown.monitoring.inHomePos AND "Unit1.Em3.ControlNodes".cmTopTapeClampTopCenterUpDown.monitoring.inHomePos AND "Unit1.Em3.ControlNodes".cmTopTapeClampTopRightUpDown.monitoring.inHomePos;
   #statTonTime[531].TON(IN := #_w1 AND "Unit1.Em3.ControlNodes".topTapeFixStage."step".transition1[531],
                         PT := T#100ms);
   IF #statTonTime[531].Q THEN
       "Unit1.Em3.ControlNodes".topTapeFixStage.sequence.status.nextStep := #JOB_5_STEP_32;
   END_IF;
END_REGION

REGION Network 40: Step[532] : Top Tape Fix Stage Bottom Clamp Down
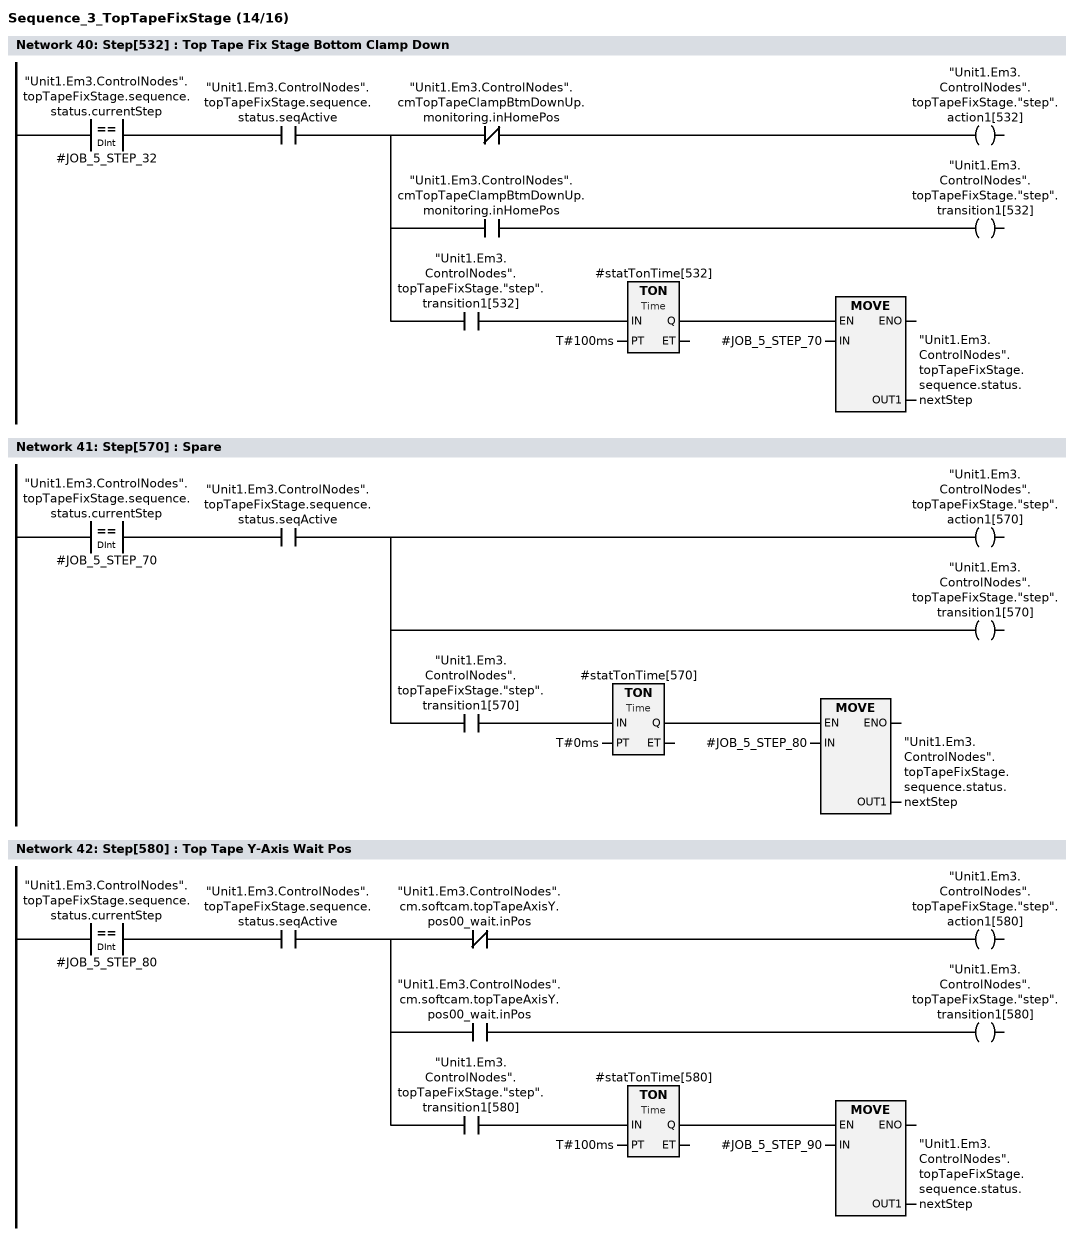
   RUNG wire#powerrail
      { S7_Templates := "SrcType := DInt" } EQ_Contact(in1 := "Unit1.Em3.ControlNodes".topTapeFixStage.sequence.status.currentStep, in2 := #JOB_5_STEP_32)
      Contact( "Unit1.Em3.ControlNodes".topTapeFixStage.sequence.status.seqActive )
      wire#w1
      I_Contact( "Unit1.Em3.ControlNodes".cmTopTapeClampBtmDownUp.monitoring.inHomePos )
      Coil( "Unit1.Em3.ControlNodes".topTapeFixStage."step".action1[532] )
   END_RUNG
   RUNG wire#w1
      Contact( "Unit1.Em3.ControlNodes".cmTopTapeClampBtmDownUp.monitoring.inHomePos )
      Coil( "Unit1.Em3.ControlNodes".topTapeFixStage."step".transition1[532] )
   END_RUNG
   RUNG wire#w1
      Contact( "Unit1.Em3.ControlNodes".topTapeFixStage."step".transition1[532] )
      { S7_Templates := "time_type := Time" } #statTonTime[532].TON(pt := T#100ms, et =>)
      Move(in := #JOB_5_STEP_70, out1 => "Unit1.Em3.ControlNodes".topTapeFixStage.sequence.status.nextStep)
   END_RUNG
   // the same network as SCL:
   #_w1 := ("Unit1.Em3.ControlNodes".topTapeFixStage.sequence.status.currentStep = #JOB_5_STEP_32) AND "Unit1.Em3.ControlNodes".topTapeFixStage.sequence.status.seqActive;
   "Unit1.Em3.ControlNodes".topTapeFixStage."step".action1[532] := #_w1 AND NOT "Unit1.Em3.ControlNodes".cmTopTapeClampBtmDownUp.monitoring.inHomePos;
   "Unit1.Em3.ControlNodes".topTapeFixStage."step".transition1[532] := #_w1 AND "Unit1.Em3.ControlNodes".cmTopTapeClampBtmDownUp.monitoring.inHomePos;
   #statTonTime[532].TON(IN := #_w1 AND "Unit1.Em3.ControlNodes".topTapeFixStage."step".transition1[532],
                         PT := T#100ms);
   IF #statTonTime[532].Q THEN
       "Unit1.Em3.ControlNodes".topTapeFixStage.sequence.status.nextStep := #JOB_5_STEP_70;
   END_IF;
END_REGION

REGION Network 41: Step[570] : Spare
   RUNG wire#powerrail
      { S7_Templates := "SrcType := DInt" } EQ_Contact(in1 := "Unit1.Em3.ControlNodes".topTapeFixStage.sequence.status.currentStep, in2 := #JOB_5_STEP_70)
      Contact( "Unit1.Em3.ControlNodes".topTapeFixStage.sequence.status.seqActive )
      wire#w1
      Coil( "Unit1.Em3.ControlNodes".topTapeFixStage."step".action1[570] )
   END_RUNG
   RUNG wire#w1
      Coil( "Unit1.Em3.ControlNodes".topTapeFixStage."step".transition1[570] )
   END_RUNG
   RUNG wire#w1
      Contact( "Unit1.Em3.ControlNodes".topTapeFixStage."step".transition1[570] )
      { S7_Templates := "time_type := Time" } #statTonTime[570].TON(pt := T#0ms, et =>)
      Move(in := #JOB_5_STEP_80, out1 => "Unit1.Em3.ControlNodes".topTapeFixStage.sequence.status.nextStep)
   END_RUNG
   // the same network as SCL:
   "Unit1.Em3.ControlNodes".topTapeFixStage."step".action1[570] := ("Unit1.Em3.ControlNodes".topTapeFixStage.sequence.status.currentStep = #JOB_5_STEP_70) AND "Unit1.Em3.ControlNodes".topTapeFixStage.sequence.status.seqActive;
   "Unit1.Em3.ControlNodes".topTapeFixStage."step".transition1[570] := ("Unit1.Em3.ControlNodes".topTapeFixStage.sequence.status.currentStep = #JOB_5_STEP_70) AND "Unit1.Em3.ControlNodes".topTapeFixStage.sequence.status.seqActive;
   #statTonTime[570].TON(IN := ("Unit1.Em3.ControlNodes".topTapeFixStage.sequence.status.currentStep = #JOB_5_STEP_70) AND "Unit1.Em3.ControlNodes".topTapeFixStage.sequence.status.seqActive AND "Unit1.Em3.ControlNodes".topTapeFixStage."step".transition1[570],
                         PT := T#0ms);
   IF #statTonTime[570].Q THEN
       "Unit1.Em3.ControlNodes".topTapeFixStage.sequence.status.nextStep := #JOB_5_STEP_80;
   END_IF;
END_REGION

REGION Network 42: Step[580] : Top Tape Y-Axis Wait Pos
   RUNG wire#powerrail
      { S7_Templates := "SrcType := DInt" } EQ_Contact(in1 := "Unit1.Em3.ControlNodes".topTapeFixStage.sequence.status.currentStep, in2 := #JOB_5_STEP_80)
      Contact( "Unit1.Em3.ControlNodes".topTapeFixStage.sequence.status.seqActive )
      wire#w1
      I_Contact( "Unit1.Em3.ControlNodes".cm.softcam.topTapeAxisY.pos00_wait.inPos )
      Coil( "Unit1.Em3.ControlNodes".topTapeFixStage."step".action1[580] )
   END_RUNG
   RUNG wire#w1
      Contact( "Unit1.Em3.ControlNodes".cm.softcam.topTapeAxisY.pos00_wait.inPos )
      Coil( "Unit1.Em3.ControlNodes".topTapeFixStage."step".transition1[580] )
   END_RUNG
   RUNG wire#w1
      Contact( "Unit1.Em3.ControlNodes".topTapeFixStage."step".transition1[580] )
      { S7_Templates := "time_type := Time" } #statTonTime[580].TON(pt := T#100ms, et =>)
      Move(in := #JOB_5_STEP_90, out1 => "Unit1.Em3.ControlNodes".topTapeFixStage.sequence.status.nextStep)
   END_RUNG
   // the same network as SCL:
   #_w1 := ("Unit1.Em3.ControlNodes".topTapeFixStage.sequence.status.currentStep = #JOB_5_STEP_80) AND "Unit1.Em3.ControlNodes".topTapeFixStage.sequence.status.seqActive;
   "Unit1.Em3.ControlNodes".topTapeFixStage."step".action1[580] := #_w1 AND NOT "Unit1.Em3.ControlNodes".cm.softcam.topTapeAxisY.pos00_wait.inPos;
   "Unit1.Em3.ControlNodes".topTapeFixStage."step".transition1[580] := #_w1 AND "Unit1.Em3.ControlNodes".cm.softcam.topTapeAxisY.pos00_wait.inPos;
   #statTonTime[580].TON(IN := #_w1 AND "Unit1.Em3.ControlNodes".topTapeFixStage."step".transition1[580],
                         PT := T#100ms);
   IF #statTonTime[580].Q THEN
       "Unit1.Em3.ControlNodes".topTapeFixStage.sequence.status.nextStep := #JOB_5_STEP_90;
   END_IF;
END_REGION

REGION Network 43: Step[590] : JOB[5] Step End
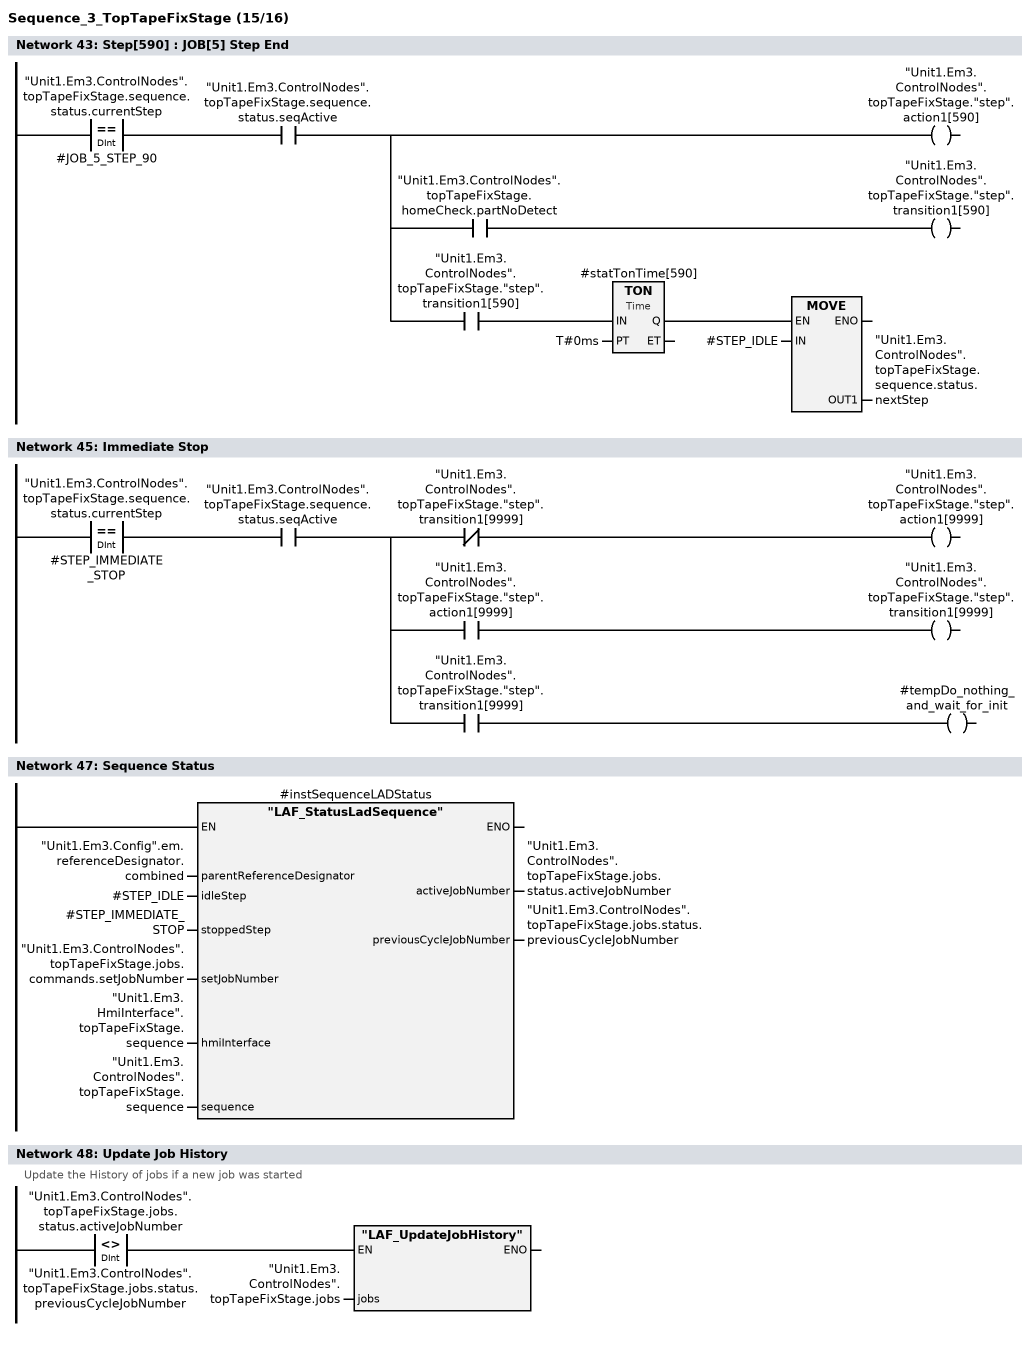
   RUNG wire#powerrail
      { S7_Templates := "SrcType := DInt" } EQ_Contact(in1 := "Unit1.Em3.ControlNodes".topTapeFixStage.sequence.status.currentStep, in2 := #JOB_5_STEP_90)
      Contact( "Unit1.Em3.ControlNodes".topTapeFixStage.sequence.status.seqActive )
      wire#w1
      Coil( "Unit1.Em3.ControlNodes".topTapeFixStage."step".action1[590] )
   END_RUNG
   RUNG wire#w1
      Contact( "Unit1.Em3.ControlNodes".topTapeFixStage.homeCheck.partNoDetect )
      Coil( "Unit1.Em3.ControlNodes".topTapeFixStage."step".transition1[590] )
   END_RUNG
   RUNG wire#w1
      Contact( "Unit1.Em3.ControlNodes".topTapeFixStage."step".transition1[590] )
      { S7_Templates := "time_type := Time" } #statTonTime[590].TON(pt := T#0ms, et =>)
      Move(in := #STEP_IDLE, out1 => "Unit1.Em3.ControlNodes".topTapeFixStage.sequence.status.nextStep)
   END_RUNG
   // the same network as SCL:
   "Unit1.Em3.ControlNodes".topTapeFixStage."step".action1[590] := ("Unit1.Em3.ControlNodes".topTapeFixStage.sequence.status.currentStep = #JOB_5_STEP_90) AND "Unit1.Em3.ControlNodes".topTapeFixStage.sequence.status.seqActive;
   "Unit1.Em3.ControlNodes".topTapeFixStage."step".transition1[590] := ("Unit1.Em3.ControlNodes".topTapeFixStage.sequence.status.currentStep = #JOB_5_STEP_90) AND "Unit1.Em3.ControlNodes".topTapeFixStage.sequence.status.seqActive AND "Unit1.Em3.ControlNodes".topTapeFixStage.homeCheck.partNoDetect;
   #statTonTime[590].TON(IN := ("Unit1.Em3.ControlNodes".topTapeFixStage.sequence.status.currentStep = #JOB_5_STEP_90) AND "Unit1.Em3.ControlNodes".topTapeFixStage.sequence.status.seqActive AND "Unit1.Em3.ControlNodes".topTapeFixStage."step".transition1[590],
                         PT := T#0ms);
   IF #statTonTime[590].Q THEN
       "Unit1.Em3.ControlNodes".topTapeFixStage.sequence.status.nextStep := #STEP_IDLE;
   END_IF;
END_REGION

REGION Network 44: *************** IMMEDIATE STOP ****************
END_REGION

REGION Network 45: Immediate Stop
   RUNG wire#powerrail
      { S7_Templates := "SrcType := DInt" } EQ_Contact(in1 := "Unit1.Em3.ControlNodes".topTapeFixStage.sequence.status.currentStep, in2 := #STEP_IMMEDIATE_STOP)
      Contact( "Unit1.Em3.ControlNodes".topTapeFixStage.sequence.status.seqActive )
      wire#w1
      I_Contact( "Unit1.Em3.ControlNodes".topTapeFixStage."step".transition1[9999] )
      Coil( "Unit1.Em3.ControlNodes".topTapeFixStage."step".action1[9999] )
   END_RUNG
   RUNG wire#w1
      Contact( "Unit1.Em3.ControlNodes".topTapeFixStage."step".action1[9999] )
      Coil( "Unit1.Em3.ControlNodes".topTapeFixStage."step".transition1[9999] )
   END_RUNG
   RUNG wire#w1
      Contact( "Unit1.Em3.ControlNodes".topTapeFixStage."step".transition1[9999] )
      Coil( #tempDo_nothing_and_wait_for_init )
   END_RUNG
   // the same network as SCL:
   #_w1 := ("Unit1.Em3.ControlNodes".topTapeFixStage.sequence.status.currentStep = #STEP_IMMEDIATE_STOP) AND "Unit1.Em3.ControlNodes".topTapeFixStage.sequence.status.seqActive;
   "Unit1.Em3.ControlNodes".topTapeFixStage."step".action1[9999] := #_w1 AND NOT "Unit1.Em3.ControlNodes".topTapeFixStage."step".transition1[9999];
   "Unit1.Em3.ControlNodes".topTapeFixStage."step".transition1[9999] := #_w1 AND "Unit1.Em3.ControlNodes".topTapeFixStage."step".action1[9999];
   #tempDo_nothing_and_wait_for_init := #_w1 AND "Unit1.Em3.ControlNodes".topTapeFixStage."step".transition1[9999];
END_REGION

REGION Network 46: *************** STATUS **********************
END_REGION

REGION Network 47: Sequence Status
   RUNG wire#powerrail
      #instSequenceLADStatus(parentReferenceDesignator := "Unit1.Em3.Config".em.referenceDesignator.combined, idleStep := #STEP_IDLE, stoppedStep := #STEP_IMMEDIATE_STOP, setJobNumber := "Unit1.Em3.ControlNodes".topTapeFixStage.jobs.commands.setJobNumber, hmiInterface := "Unit1.Em3.HmiInterface".topTapeFixStage.sequence, sequence := "Unit1.Em3.ControlNodes".topTapeFixStage.sequence, activeJobNumber => "Unit1.Em3.ControlNodes".topTapeFixStage.jobs.status.activeJobNumber, previousCycleJobNumber => "Unit1.Em3.ControlNodes".topTapeFixStage.jobs.status.previousCycleJobNumber)
   END_RUNG
   // the same network as SCL:
   #instSequenceLADStatus(parentReferenceDesignator := "Unit1.Em3.Config".em.referenceDesignator.combined,   // "LAF_StatusLadSequence"
                          idleStep := #STEP_IDLE,
                          stoppedStep := #STEP_IMMEDIATE_STOP,
                          setJobNumber := "Unit1.Em3.ControlNodes".topTapeFixStage.jobs.commands.setJobNumber,
                          hmiInterface := "Unit1.Em3.HmiInterface".topTapeFixStage.sequence,
                          sequence := "Unit1.Em3.ControlNodes".topTapeFixStage.sequence,
                          activeJobNumber => "Unit1.Em3.ControlNodes".topTapeFixStage.jobs.status.activeJobNumber,
                          previousCycleJobNumber => "Unit1.Em3.ControlNodes".topTapeFixStage.jobs.status.previousCycleJobNumber);
END_REGION

REGION Network 48: Update Job History
   // Update the History of jobs if a new job was started
   RUNG wire#powerrail
      { S7_Templates := "SrcType := DInt" } NE_Contact(in1 := "Unit1.Em3.ControlNodes".topTapeFixStage.jobs.status.activeJobNumber, in2 := "Unit1.Em3.ControlNodes".topTapeFixStage.jobs.status.previousCycleJobNumber)
      "LAF_UpdateJobHistory"(jobs := "Unit1.Em3.ControlNodes".topTapeFixStage.jobs)
   END_RUNG
   // the same network as SCL:
   IF "Unit1.Em3.ControlNodes".topTapeFixStage.jobs.status.activeJobNumber <> "Unit1.Em3.ControlNodes".topTapeFixStage.jobs.status.previousCycleJobNumber THEN
       "LAF_UpdateJobHistory"(jobs := "Unit1.Em3.ControlNodes".topTapeFixStage.jobs);
   END_IF;
END_REGION

REGION Network 49: Output steps as String
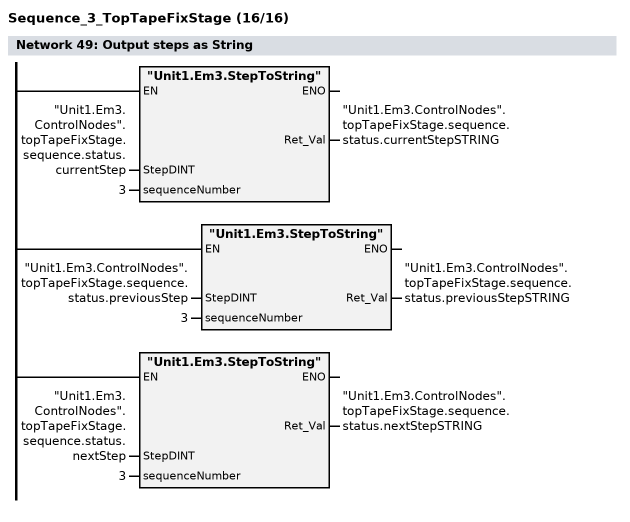
   RUNG wire#powerrail
      "Unit1.Em3.StepToString"(StepDINT := "Unit1.Em3.ControlNodes".topTapeFixStage.sequence.status.currentStep, sequenceNumber := 3, Ret_Val => "Unit1.Em3.ControlNodes".topTapeFixStage.sequence.status.currentStepSTRING)
   END_RUNG
   RUNG wire#powerrail
      "Unit1.Em3.StepToString"(StepDINT := "Unit1.Em3.ControlNodes".topTapeFixStage.sequence.status.previousStep, sequenceNumber := 3, Ret_Val => "Unit1.Em3.ControlNodes".topTapeFixStage.sequence.status.previousStepSTRING)
   END_RUNG
   RUNG wire#powerrail
      "Unit1.Em3.StepToString"(StepDINT := "Unit1.Em3.ControlNodes".topTapeFixStage.sequence.status.nextStep, sequenceNumber := 3, Ret_Val => "Unit1.Em3.ControlNodes".topTapeFixStage.sequence.status.nextStepSTRING)
   END_RUNG
   // the same network as SCL:
   "Unit1.Em3.ControlNodes".topTapeFixStage.sequence.status.currentStepSTRING := "Unit1.Em3.StepToString"(StepDINT := "Unit1.Em3.ControlNodes".topTapeFixStage.sequence.status.currentStep,
                           sequenceNumber := 3);
   "Unit1.Em3.ControlNodes".topTapeFixStage.sequence.status.previousStepSTRING := "Unit1.Em3.StepToString"(StepDINT := "Unit1.Em3.ControlNodes".topTapeFixStage.sequence.status.previousStep,
                           sequenceNumber := 3);
   "Unit1.Em3.ControlNodes".topTapeFixStage.sequence.status.nextStepSTRING := "Unit1.Em3.StepToString"(StepDINT := "Unit1.Em3.ControlNodes".topTapeFixStage.sequence.status.nextStep,
                           sequenceNumber := 3);
END_REGION
END_FUNCTION_BLOCK
